(* IEC 61131-3 sources: ml2plc/benchmarks/st (part 22) *)

(* ---- ResNet3.st ---- *)
FUNCTION_BLOCK ResNet3_FB

    (* Model Inputs/Outputs *)
VAR_INPUT
    input_data : REAL;
END_VAR

VAR_OUTPUT
    output_data : ARRAY[0..2] OF REAL;
END_VAR

VAR CONSTANT
    weights_0 : ARRAY[0..63] OF REAL := [-0.190466672, -0.289495766, 0.36445868, 0.11001166, -0.202885658, -0.247976601, -0.217859656, 0.152941793, -0.210685372, 0.322490484, -0.300406843, -0.0737419277, 0.271309823, 0.34986949, -0.269151628, 0.101570874, -0.0975821763, -0.0239237547, -0.28141278, -0.260361493, 0.220720425, 0.342909008, -0.106619239, 0.192217126, -0.139923915, -0.00473925471, 0.256588012, 0.106521919, -0.015166074, -0.237258494, -0.295479923, 0.237283707, -0.111313865, -0.119793385, -0.189164549, 0.109231912, 0.147311017, -0.0809866935, -0.174528345, -0.015255332, 0.110069647, 0.205406636, 0.233189464, 0.175904229, 0.192441761, -0.257080823, 0.113344185, -0.222640619, 0.0253927261, -0.0698330998, 0.304976135, 0.13343668, -0.229343772, 0.317507595, -0.0133918505, 0.251467377, -0.131539866, -0.128968731, 0.204563618, -0.234828115, 0.109687969, 0.0967651531, -0.128085941, 0.0570141077];
    bias_0 : ARRAY[0..63] OF REAL := [0, 0, -0.0451503769, -0.000170675936, 0, 0, 0, -0.0306519736, 0, -0.043658372, 0, 0, -0.0452437028, -0.0463685207, 0, -0.0237470753, 0, 0, 0, 0, -0.0306253415, -0.0182554778, 0, -0.0286273304, 0, 0, -0.0439416394, 0.0359471515, 0, 0, 0, -0.0393987, 0, 0, 0, -0.025377661, 0.0258860644, 0, 0, 0, -0.0256011337, -0.040137399, -0.0210138671, -0.0197667424, -0.0420954861, 0, -0.0343104228, 0, -0.0101194074, 0, -0.0385119878, -0.0309600942, 0, -0.0221530851, 0.0427107885, -0.0482655875, 0, 0, -0.0332414694, 0, -0.0204843841, -0.0293239169, 0, -0.0204854961];

    weights_1 : ARRAY[0..4095] OF REAL := [-0.0287969261, 0.201637134, -0.193626225, -0.0838745981, -0.179824859, -0.158866256, -0.0519343764, 0.0553617924, -0.0298234671, 0.199577436, -0.0565214604, -0.135609776, 0.19474043, -0.0305772722, 0.047594741, 0.174586251, -0.131670237, -0.0606977493, -0.00999130309, 0.160562769, 0.114603773, 0.198183253, -0.0226515681, -0.174445733, 0.0844327062, -0.0653743893, 0.166338369, 0.178600982, -0.179540232, -0.104543671, -0.04106462, 0.0376635343, -0.0928359851, 0.0239627361, -0.0751802325, -0.131423861, 0.107191309, 0.0680955499, -0.134543836, 0.162752822, -0.119452722, -0.118079856, -0.111446388, 0.103158936, -0.0164598525, -0.143377468, 0.0849187821, -0.0122491121, -0.152280733, -0.120597631, -0.0606369525, -0.0807449222, 0.147399679, 0.0629173666, -0.130655468, -0.21262382, -0.169020504, 0.105712339, 0.11746116, 0.0592246503, -0.0597587526, -0.143656209, 0.0653275698, -0.0477767587, -0.154527515, 0.0485876948, -0.0317480415, -0.000382602215, -0.0967821628, 0.0423714072, -0.0512648225, 0.0312831551, -0.17014426, 0.160105124, 0.109350279, -0.0217197388, -0.0921072736, 0.0853802711, -0.0300633907, 0.135347292, -0.0391751528, -0.199345261, -0.195168182, 0.0560685545, 0.215828583, -0.0923638716, 0.192498907, 0.178375289, -0.183688045, 0.116588429, 0.0289125443, 0.0778251439, 0.0613025278, 0.0142809004, 0.0337732583, 0.0574108511, 0.189165697, 0.196946517, 0.107737496, -0.129702166, -0.107477285, -0.107738689, -0.177952528, -0.0559140593, 0.169283316, -0.0538910031, -0.104346119, -0.127213195, -0.0331750959, 0.127317414, 0.0515208095, 0.0195653588, 0.0769012719, -0.124866173, 0.177239373, 0.0280220658, 0.0963039249, -0.0652452409, 0.105720118, 0.15663074, -0.136386782, -0.123085879, 0.0827278346, 0.21160166, -0.16991207, -0.0768297166, 0.120611772, 0.134732291, -0.139711812, -0.184518486, -0.184835598, 0.00858225208, 0.113042273, -0.102391459, -0.0780269504, -0.165388852, -0.140612379, 0.223779544, 0.162238076, -0.00674940646, 0.0487292968, 0.0836367309, -0.19456315, 0.171644017, -0.0955267325, 0.0997560844, -0.0601457544, -0.198954478, -0.00482972385, -0.079228431, -0.127536789, 0.190665379, -0.0999609306, 0.0110752583, -4.10255961e-05, 0.118868679, 0.138081178, -0.0528386459, -0.114722773, 0.170001924, 0.137378082, -0.196978897, -0.15748626, 0.0825704783, -0.033234071, -0.101335384, 0.0289265234, -0.15857622, -0.0556612536, 0.213226333, 0.00719815027, 0.223965615, -0.0638628826, 0.148281991, 0.0975444093, -0.0259753708, 0.0262751374, 0.0979252607, -0.0863377675, 0.0899253041, 0.239503771, 0.289376885, -0.204818711, 0.105383582, 0.293127954, 0.203753337, -0.119700439, -0.16846402, 0.191751063, 0.0327624083, -0.0386312976, -0.264414817, 0.153028056, 0.154591411, 0.124344207, -0.107223384, -0.137165904, 0.0300747007, 0.183606654, 0.198948666, 0.0499654785, 0.144469813, -0.210293442, -0.0324280113, 0.0683567002, -0.04100243, -0.0126516968, 0.164788797, 0.237893194, -0.0847178176, 0.0626023933, 0.155760348, 0.185824335, 0.00780587131, 0.199899733, 0.035005752, -0.0749012083, 0.067025587, 0.141089186, -0.0444214866, -0.0607198402, 0.0990498737, -0.0620695017, 0.0086689936, -0.114031576, -0.111011893, -0.204213917, -0.198096737, 0.138905957, 0.159203395, 0.12167336, 0.0172255039, 0.15101482, 0.131718054, -0.0235928968, 0.200807258, 0.209497362, 0.170748204, -0.231670231, 0.143206522, 0.225486189, 0.104716703, -0.177130625, -0.133289889, -0.0483859442, 0.107198499, -0.0196592454, -0.0476846471, -0.0815907568, -0.135093376, 0.12207596, 0.00658966927, -0.0573140644, 0.0118645504, 0.226763472, 0.178059682, -0.0891532153, 0.0825275332, 0.163484469, -0.0550447851, -0.0375959724, -0.00878846645, 0.0168165267, 0.150091812, 0.084491238, 0.174592748, 0.0785937458, 0.163301513, -0.0316622555, 0.0597050637, 0.157956466, -0.0453870595, 0.101291135, -0.0735865831, 0.0523432046, 0.00310024619, -0.111143999, -0.176621795, 0.0883997232, -0.00594709814, -0.0267459899, 0.164880231, 0.0904007405, -0.00336711109, 0.025017634, -0.136061743, -0.0808758289, 0.139091626, 0.0775778443, -0.155642897, 0.0725118369, -0.0960384831, 0.135437921, -0.188861921, 0.0681308657, 0.121807054, -0.0181216151, 0.126562431, 0.0201322883, 0.0685440749, 0.0470108241, 0.206563786, 0.167886898, -0.182285488, -0.166398615, 0.200898841, 0.191317186, 0.190035328, -0.175405696, 0.124712333, 0.052170679, 0.184364364, -0.0736751109, 0.0639937371, -0.168305129, 0.00677789748, -0.148140043, 0.10284771, -0.13430731, 0.139501527, 0.0359104425, 0.0577303618, -0.188823983, -0.174651235, 0.0696652383, -0.183670074, -0.00257234275, -0.193130046, -0.203748837, -0.153786868, 0.202487156, -0.0460375547, 0.109957233, 0.00299288332, -0.162598059, 0.210710511, -0.194323435, -0.210184813, 0.0554226786, -0.142163336, -0.152110279, -0.0163246542, -0.166943565, 0.175032482, -0.215747178, 0.171988502, 0.132436678, 0.172353908, 0.121031687, 0.186095968, -0.0588158816, -0.0108129233, -0.0942323804, -0.09778703, -0.109081298, -0.106757924, 0.172346756, 0.025905624, 0.0740813166, 0.189657524, 0.148814008, 0.197771326, 0.201267496, -0.068178758, 0.1481594, 0.184583381, -0.014007479, 0.0497234613, -0.0900920182, -0.151112944, -0.154349625, 0.155235782, -0.183371142, -0.164333746, 0.110023871, 0.0927015692, 0.194937959, 0.208203807, -0.00641842186, -0.135277599, -0.0120722651, 0.0209348053, -0.163213924, 0.183399543, 0.00101952255, -0.094531931, -0.0417330861, 0.125320569, 0.140007362, -0.0551816374, -0.0750101358, -0.184187144, 0.0996663719, 0.1298704, -0.00832244754, -0.00248210132, 0.0548401624, -0.0217346549, -0.040534541, 0.0774618536, 0.0789829642, -0.213013336, 0.00969907641, 0.131764188, -0.134339929, -0.16999869, -0.150505453, -0.203993306, 0.133900389, 0.210885063, 0.0592023879, 0.119564161, 0.129766181, -0.116630182, 0.0890186876, 0.0916796774, -0.125102013, 0.144167438, 0.190863922, 0.0828631073, 0.110106811, -0.0818011016, 0.0638723224, 0.0225199312, -0.0798923373, -0.106765099, -0.103232488, -0.0746515393, 0.214082971, -0.139221311, 0.0676382631, 0.20862554, 0.185882255, -0.0279404521, 0.0581518859, -0.0932726786, -0.0684341788, -0.148790196, -0.167229846, 0.160150275, -0.125400275, -0.0166903287, -0.0369179547, 0.0845469385, -0.191490114, -0.161978155, -0.023997426, 0.040678516, 0.14639619, 0.0431083404, 0.0106931906, 0.139329195, -0.149284765, -0.0467167646, -0.0767225027, -0.0320999771, -0.23229675, -0.0372863598, 0.128295347, -0.160325885, -0.148059294, -0.00792731252, 0.0252128541, -0.0963003412, -0.0197790675, -0.0523058102, -0.0141548719, -0.168405354, 0.093509756, -0.0733992159, -0.174149796, 0.0823272243, 0.0543129146, 0.00202205591, 0.112447657, -0.189444944, 0.0949934795, 0.133855537, 0.138600275, -0.170810059, -0.0500965714, -0.186440244, 0.0285257101, -0.000778779387, -0.128126383, -0.0261946935, -0.201500729, 0.11489366, 0.0997269675, -0.138657212, -0.256732196, 0.0291550159, -0.302546233, -0.178278208, -0.234763011, -0.0388856418, 0.0533248745, -0.146624878, -0.0823597312, -0.230229869, 0.0182416849, -0.118736058, 0.0481926613, 0.133541629, -0.114781246, 0.10070549, 0.109701976, 0.0569074266, 0.26510939, 0.00950349867, 0.0546200871, 0.151336238, 0.0048430115, 0.0378029197, 0.144169971, 0.0863773972, 0.200766638, 0.212797061, 0.138086304, -0.182377681, 0.213811055, 0.161403164, 0.124502376, 0.0246564448, -0.196184307, -0.196561068, 0.0875730366, 0.0948206931, -0.149286091, 0.0323978215, 0.0455216914, 0.151648596, -0.127112329, -0.111039624, 0.0246137083, 0.016291365, -0.00267861784, 0.0558695644, 0.201473311, -0.178703129, -0.103530645, 0.173463836, 0.157130465, 0.182277635, 0.0760518163, 0.215445682, -0.106563114, -0.196684077, -0.094135493, 0.10404627, 0.0962792784, -0.0124557465, -0.15429759, -0.0716400295, 0.11189805, 0.0764795393, 0.0549422354, -0.0472201556, -0.00484439731, 0.0528673977, 0.190446272, 0.0174336433, -0.0469030589, -0.0549324602, 0.102302983, -4.00096178e-05, 0.147421315, 0.193782583, -0.0265746713, 0.0705426186, 0.0295248479, -0.134114474, 0.0562623292, 0.172508165, 0.175126389, -0.161904559, -0.0162163712, 0.208393365, -0.100752503, 0.0273437109, -0.153811902, -0.193232462, -0.16940017, 0.188474581, -0.0369768888, 0.0354307853, -0.0991368741, -0.196591377, -0.233054638, -0.118758805, -0.0622535497, 0.0394661725, 0.267733514, 0.107220888, -0.252435923, 0.112368457, 0.166412622, 0.192772374, -0.218732044, 0.126407787, 0.0919501036, 0.00824039057, -0.0796734989, 0.182596043, 0.131103203, -0.109326825, 0.125145733, 0.122357175, 0.0696524829, -0.0965674892, 0.0579061955, -0.200026214, -0.185237691, -0.189040273, -0.224097118, 0.103700139, 0.109744169, 0.283211142, -0.108721465, 0.126635522, -0.0494364649, -0.224469841, 0.151249424, -0.162036136, 0.030354334, -0.00598688424, -0.143472508, -0.047887668, 0.0439753979, 0.0527719408, -0.152598977, 0.110804304, 0.257972151, -0.138091505, -0.110594928, 0.100734361, -0.0214415565, 0.0449742526, 0.22822006, -0.240381643, -0.128085867, -0.0693219751, -0.0846015364, -0.17030485, 0.130928531, 0.00229240954, -0.194736332, -0.0391959101, 0.0145413131, -0.144774944, -0.181710035, 0.032208994, -0.206829414, -0.0198655725, 0.0611966401, 0.00840911269, 0.158986792, 0.126695439, -0.157956257, -0.20029664, -0.104722835, -0.144183606, 0.00487022102, 0.0939430147, -0.0584943891, 0.0557004064, 0.00045491755, 0.114710584, 0.0546646267, 0.20419623, 0.0921241492, 0.0991390496, 0.176430956, -0.158750683, -0.0890071839, -0.179640472, 0.162403598, -0.0909959227, 0.0409451872, -0.0232819319, 0.165903732, 0.069598332, 0.175637826, -0.179648638, -0.00545862317, 0.00749818981, 0.0323755145, -0.158800021, 0.180631563, -0.053162545, -0.014888972, -0.188607126, -0.0488055795, 0.20547007, -0.0377693027, 0.0997820646, -0.124526724, -0.0918210968, -0.167447731, -0.188922942, 0.0540182441, 0.122466967, -0.0612903982, 0.173171565, 0.187880501, 0.0320709199, -0.0716537684, -0.146939963, 0.00549939275, 0.0170418024, -0.156284317, -0.158158392, -0.0161726922, -0.117838174, 0.0458692163, 0.0690316111, -0.102591947, -0.0113369077, -0.0506339818, 0.186475053, 0.10736011, -0.0328097939, -0.13072902, -0.14560762, 0.0873160809, 0.204848334, 0.079661116, -0.018868804, -0.018476963, 0.148941293, 0.0539769381, -0.00221420825, -0.108419128, -0.0766489506, -0.189365566, 0.0919391662, -0.212484032, -0.172094896, 0.0239589214, -0.211048037, 0.189641103, 0.0730664879, 0.206356838, -0.135675371, -0.000756576657, 0.0285059959, 0.209358588, 0.192232445, 0.11306645, -0.115133278, 0.175952092, 0.0211753547, 0.0506318063, -0.19809112, 0.0197272301, 0.054157868, 0.0254253149, -0.155184671, -0.0454918444, -0.196502686, -0.0158347338, -0.135656744, -0.211595923, -0.020885095, -0.00690788031, 0.0370714217, -0.172456279, -0.185076281, 0.160629585, 0.0181837529, -0.0211855043, 0.120963901, -0.00527728582, -0.0352699608, -0.19402647, 0.132209137, 0.0396415927, -0.118135475, 0.00657442212, -0.208759815, -0.0303688291, -0.00777827017, -0.0915059149, 0.11210835, 0.294361055, -0.142053381, -0.0571834072, -0.0146589978, -0.0864291564, -0.101504333, 0.12920031, 0.182926923, 0.192566365, 0.106406614, 0.214629248, 0.06889496, -0.11516425, -0.259321928, 0.184162751, -0.272702873, -0.117973782, 0.0606180206, 0.0292263925, 0.0766455382, -0.120667271, -0.201999113, -0.0266232025, -0.00732299685, -0.0519965291, 0.156876504, 0.123033859, 0.267217845, -0.0109749781, -0.272964209, -0.129237577, 0.053774897, 0.141416252, -0.199857935, 0.0538020581, -0.230259433, -0.0451727808, 0.258897543, 0.148216307, -0.053409934, 0.31615606, 0.0147380829, -0.202499956, 0.110624768, 0.1696845, -0.0922751948, 0.0798982531, 0.0207011886, -0.142718717, 0.0519616678, -0.127546012, 0.126492023, 0.0723542273, 0.147747502, 0.126169741, 0.0813353807, -0.1203655, -0.153749913, -0.0919978395, -0.139003664, 0.0844179541, 0.054092221, 0.110275611, -0.200139761, 0.110008813, -0.126036033, -0.166970596, -0.233972371, 0.0890860558, -0.20025298, -0.230093077, 0.0173213258, 0.275560528, 0.151483357, 0.276097506, 0.00718977815, -0.0111169517, 0.168895632, 0.10235633, -0.240326077, -0.0821303874, -0.00890312064, -0.171553358, -0.00546233356, 0.101003714, 0.0433369204, -0.187788144, -0.103547342, 0.00432489906, -0.109544538, 0.012347714, 0.0869178474, -0.257481515, -0.0600075051, -0.264836371, -0.171154037, 0.0307734851, -0.129194021, -0.199388355, 0.0987441167, -0.0623329841, 0.249395654, -0.034193743, 0.0902072638, 0.203402102, -0.0227374583, 0.0134097785, -0.0912396759, 0.0864051133, 0.0865284353, 0.228083283, 0.126239121, -0.109470509, -0.188946784, 0.00514312088, 0.181860104, 0.0482862443, 0.0316015482, 0.208089277, 0.175173715, 0.157937661, -0.175959155, -0.15175122, 0.0449968129, -0.0724449754, 0.131373897, 0.081098035, 0.0556937009, -0.127380341, 0.131804869, -0.182943538, -0.163977832, -0.00456343591, 0.0986122638, -0.0509269685, 0.144946262, 0.152006164, -0.195760101, -0.158920705, -0.0407915562, 0.0382466763, 0.120302364, 0.163731501, 0.0790192336, 0.0871210247, -0.0502094626, -0.193163037, 0.0618805438, -0.0852957666, 0.124724433, 0.0312432498, 0.114015713, 0.150832668, 0.00696192682, -0.020202592, 0.0919532925, 0.0599388927, -0.155759037, -0.0923569575, -0.0696199685, -0.127464831, -0.187969327, -0.187459841, 0.143950805, -0.0970960557, 0.154307649, -0.05652605, 0.156533435, -0.183348998, 0.139695272, 0.124307856, -0.0476845652, 0.0955802649, -0.0311176628, 0.163419768, 0.113613471, 0.182277307, -0.202524781, 0.0122317718, 0.186174095, -0.113051899, 0.208240613, -0.158425584, 0.0850085169, -0.0775510222, -0.0645689219, -0.0517540723, -0.17061533, 0.0819323882, 0.121917769, -0.119305968, -0.0747042894, 0.0523318127, -0.152910829, 0.100246899, 0.0908019319, 0.066256009, -0.0805988908, 0.0907654166, 0.0451934189, -0.0514816083, 0.192991301, 0.180941716, -0.197929591, -0.0896847397, -0.218640536, 0.058635354, -0.112284772, -0.0678162426, -0.0591657534, 0.190862313, -0.0746522695, -0.0959051773, -0.0859087706, 0.0146463895, 0.127395496, 0.0643470958, 0.222248226, -0.222716317, -0.0038960767, 0.0420699306, -0.189540833, 0.151158154, 0.174533531, 0.0537843928, 0.0724432617, -0.0636890829, -0.0554191582, 0.0796529651, 0.220607117, -0.152003556, 0.0678689852, 0.189509705, 0.196022376, 0.112115934, -0.103596382, 0.0718052611, -0.139615148, 0.17220287, -0.108806856, -0.0700540841, -0.126261801, -0.0981526002, -0.0755177587, 0.112252161, 0.196778193, -0.00826221704, -0.185675785, -0.057513833, -0.101335384, 0.0925282687, -0.0817712694, -0.131041422, -0.0185560435, -0.125542641, 0.191311106, 0.183952644, 0.13196452, -0.153428495, -0.117309444, -0.0829459131, -0.110064179, 0.198635712, -0.171391279, 0.111330763, -0.148759633, 0.0993963033, 0.0926398188, 0.208881006, 0.106514856, 0.205308661, 0.0648586303, 0.000817343593, -0.0404887646, 0.129113868, -0.0304635465, 0.057734862, -0.0244514644, 0.102735177, 0.120236859, -0.138929337, 0.0624369532, -0.155432343, -0.15313834, 0.0859217495, -0.00519438088, 0.126614913, -0.21491994, 0.0207336992, 0.175207987, 0.109249786, -0.054661721, 0.0479473621, 0.00943541527, -0.142473519, 0.116482362, 0.0937203616, -0.0977497622, 0.183454707, 0.126636133, 0.132889017, -0.179818153, -0.00318422914, -0.114538781, 0.190620884, -0.0922307968, 0.171573177, -0.113899581, 0.0264129937, -0.117907241, 0.0159941912, 0.056949541, -0.165546909, -0.079548344, 0.155183807, 0.167912915, -0.12471018, -0.0227756053, 0.195206597, 0.155959591, -0.113060772, 0.0471404046, -0.0937578529, -0.0744760931, 0.0718369633, -0.194636658, 0.0701943189, 0.00457412004, -0.0688510537, -0.159001023, 0.119077131, 0.0420625359, -0.101866595, -0.0260792822, -0.213209078, -0.0761060715, 0.0378767401, -0.0494340956, 0.0950354189, -0.119263433, -0.187393367, -0.19390738, -0.115837008, -0.11679624, 0.0311641246, -0.0763715953, 0.00562612712, 0.104230031, -0.0938740447, -0.158894032, -0.186505824, 0.123571053, 0.0021596998, -0.124141335, 0.0726272911, 0.0728365034, 0.048231259, 0.167245731, 0.173797145, -0.133879036, 0.123410001, 0.0136341602, 0.211613938, 0.0339705497, -0.0568555892, -0.0638442487, -0.165108442, 0.113140717, -0.114156596, 0.0502677411, 0.105490163, 0.154489145, 0.0633081943, 0.0605547279, -0.168472469, -0.174018279, -0.178102687, -0.0923157632, 0.0868086368, 0.142751232, 0.0472065359, -0.0355895907, -0.070602119, 0.0226132125, 0.111900166, 0.072677359, 0.126415685, -0.147081137, -0.145128071, 0.119609222, -0.149196088, -0.0602950752, 0.198493585, 0.137908891, 0.0641960949, 0.200968578, -0.0566390008, -0.1688862, 0.172993645, -0.144077167, -0.197343826, -0.0247414112, 0.199622199, -0.1655339, -0.0133733898, 0.134934023, 0.0719420165, 0.000706866384, 0.149509206, -0.156804532, -0.0837745517, -0.037465632, -0.157091066, 0.107307032, -0.00644093752, 0.0704480559, -0.183203697, -0.196138009, -0.117853299, -0.12040215, -0.11014574, -0.116727851, 0.026737988, -0.0404386818, 0.0639270395, 0.104571596, 0.0609508008, -0.0830935389, -0.20587337, 0.0998597592, 0.0920080096, -0.113937676, -0.0127168447, 0.130367443, -0.162072524, 0.206473872, -0.0470631719, 0.202682182, -0.0224076658, -0.0183282048, -0.0392407626, 0.13104786, 0.0124193132, -0.155867845, 0.187796101, 0.12736474, 0.183426574, 0.0451046377, 0.0507078916, 0.122980073, -0.21496205, 0.0355659574, -0.0358312726, -0.136690676, -0.167069823, 0.0553592891, 0.212405875, 0.186634675, 0.140052691, 0.0532232374, -0.132964134, 0.199990019, 0.129920498, -0.0277204067, 0.162883624, 0.197279349, -0.0547595471, -0.169750974, -0.0363512784, -0.0266377479, 0.122363672, 0.0337654799, -0.199149102, 0.207519457, 0.142926887, 0.215468749, -0.0605023801, -0.0568595082, 0.0636674613, 0.106427982, -0.139160648, -0.11427062, 0.189653918, 0.135131165, -0.0713291317, 0.103454813, 0.115515873, 0.0241415501, -0.141884476, 0.0647414476, 0.1221935, 0.187437966, -0.0765461177, 0.130906656, 0.209548905, 0.198075101, -0.0151947271, 0.106877655, 0.122374028, 0.0876808092, -0.0646020845, 0.179015324, 0.137440547, -0.111645944, -0.0637109131, 0.264909327, -0.00986942649, 0.19460775, -0.215875, -0.216673881, -0.195247158, 0.0369132459, 0.22958532, -0.0758189484, 0.161118656, -0.0532057211, -0.111272402, 0.0191001799, 0.154950529, 0.184459001, -0.0586241372, 0.211076126, 0.0385005176, 0.0375854224, 0.185866401, -0.0925790668, 0.0594946295, -0.199379593, 0.160706773, -0.0215413142, 0.0920865387, -0.0727619678, -0.0503336526, 0.144037127, 0.0390647538, -0.176736578, 0.218084648, 0.282077163, 0.0684015825, -0.0997406542, 0.0936136246, -0.0177756548, -0.116294734, -0.21881853, 0.0861533135, -0.144913971, -0.116913833, -0.228465006, 0.243279889, 0.289645553, -0.157389015, 0.0694431514, -0.0845005885, -0.169205248, 0.0732500702, -0.140289873, 0.217532694, -0.153820172, 0.165036872, -0.0370052084, -0.0649239048, 0.00705603603, 0.00300642545, -0.147408083, -0.0400309153, -0.0219824761, 0.021092033, -0.0739108026, 0.0152327912, 0.16345866, -0.169258162, -0.171906739, -0.0344251506, 0.0626144186, 0.0827743858, 0.0153012248, 0.214705959, 0.149533838, -0.0852295235, 0.108769022, -0.125927284, 0.0506657287, -0.0685000271, 0.132542357, 0.189130142, -0.107204311, 0.208437741, -0.0613691844, -0.15225552, 0.0756992996, -0.0966535062, -0.198031753, 0.0743363649, 0.0633449629, -0.129061252, 0.122365281, -0.130634353, 0.0883900598, 0.0156343877, -0.135135397, 0.198845685, 0.2392952, -0.145629406, 0.188295275, -0.13789998, 0.132967234, 0.132922307, -0.17668727, 0.245915323, -0.141065955, 0.192191795, -0.157576233, -0.085805878, -0.0276803467, -0.095566079, 0.219359696, 0.202878788, -0.0802682042, -0.176504254, 0.023325054, 0.0037062054, -0.138832927, 0.053536851, 0.127934501, -0.168392971, 0.0300281346, 0.0400527865, -0.206524342, -0.081766516, 0.104110494, 0.00106944144, -0.120554268, -0.0580964088, 0.109146222, -0.000105708838, 0.182546988, -0.148469537, -0.148119092, 0.149815395, 0.205082461, -0.0108131766, 0.179644182, -0.192448467, -0.0218183249, 0.112928316, 0.173357442, 0.0719634742, 0.20145084, 0.0719409138, -0.164568782, -0.130916566, -0.202400431, 0.0947056264, -0.192789838, 0.0868111402, -0.00978286564, 0.196489051, -0.0734990388, -0.146960199, -0.000552743673, 0.0167299211, -0.199335337, -0.158682853, 0.0911645144, 0.180834278, -0.122386955, 0.00548417866, -0.187905684, -0.107697234, -0.084947437, 0.0716611892, 0.132587507, 0.13105391, 0.0321043134, 0.0708666295, 0.136131003, 0.0918786675, 0.0526147634, 0.14389886, -0.0311155468, -0.188370556, -0.212843508, 0.0522523373, 0.167048857, -0.206337899, 0.072918728, 0.120494351, -0.190175474, -0.154683962, -0.000773754495, -0.186758995, 0.25392881, 0.165069968, -0.174278378, -0.0480074361, 0.0444551259, -0.0307127461, 0.197782025, 0.127323076, -0.19140029, -0.17637898, -0.0651647598, -0.0631855875, -0.170364678, 0.128072217, 0.142127141, 0.0896252617, -0.168872684, 0.0608825311, -0.199593708, 0.0163794793, -0.111544512, -0.0925613791, 0.0456584245, 0.273554981, 0.0908730105, -0.121767685, 0.133312061, -0.0430089869, 0.048706051, -0.106118105, 0.156891361, 0.199550763, 0.0661296993, 0.190545216, 0.0400548801, 0.0303085539, -0.0425427854, 0.0662297159, 0.266184568, 0.028025724, -0.122740746, 0.0264457632, 0.00358478306, 0.129521757, 0.162871301, 0.26886633, -0.0782814473, -0.0386863798, -0.0817479417, 0.0508834422, 0.212506562, -0.104619637, 0.0130023751, 0.0292652808, -0.08503066, 0.158758327, 0.0168799069, -0.0856374726, -0.150301456, -0.0860033929, -0.118447781, -0.179989219, -0.0929494426, -0.0466621518, -0.0659421533, 0.121023342, 0.105154112, -0.0455614179, -0.203972697, 0.173838392, -0.0386415124, -0.0278328806, 0.178764507, 0.104911312, 0.108715996, -0.0253986865, -0.168122798, -0.114805967, -0.0621888191, -0.0132009238, 0.0253832936, -0.0265160799, 0.0423865467, -0.100953348, 0.172172591, 0.201425806, 0.141991392, 0.0940631181, 0.194293097, 0.0401813537, 0.12128751, 0.196684197, -0.0543928444, 0.0463825911, 0.0403407067, -0.21529898, 0.00518736243, -0.0455965251, 0.0162204355, -0.183138445, -0.193831608, 0.187192395, 0.00752931833, 0.157815233, 0.141796991, -0.0405156463, 0.198203638, 0.00560341775, -0.0508095473, -0.0763344318, -0.0735320747, -0.0695720166, 0.148685709, 0.0700013191, 0.182473376, -0.1108841, -0.0968367755, 0.0362190455, 0.036774829, 0.0170685947, -0.0752303004, -0.0852943808, -0.206426427, -0.149846435, -0.155158252, 0.119575307, 0.0180834234, 0.146422639, -0.101406202, 0.0536810011, 0.0994656831, -0.0630992353, 0.0158559978, -0.0455258042, -0.21185334, -0.118426792, 0.159210399, -0.116417825, 0.0386347026, 0.159501418, 0.033601746, -0.0757299215, 0.00185963511, 0.085397765, 0.083639726, 0.178043649, 0.190545216, -0.0945898443, 0.0499521047, 0.0201606303, 0.106833711, -0.0188183188, 0.177461788, -0.100810207, -0.0469589531, -0.0987466872, 0.177121416, 0.1593398, 0.0223871171, -0.208162114, 0.062356934, -0.125736207, 0.096315518, 0.0971169025, 0.0245347768, -0.020675838, -0.111754142, 0.212888882, -0.170801476, 0.0786470622, -0.0122303218, 0.162038699, -0.199096397, 0.170362726, 0.0747093409, 0.111208364, -0.0473197848, -0.0435504466, -0.0453317761, -0.110917084, -0.0126232058, -0.177978754, -0.0992414504, 0.130278543, 0.018110469, -0.0700823665, -0.114136361, 0.0361899287, -0.18268013, 0.0165710393, 0.0793500915, -0.00841967668, 0.125138253, 0.0887469351, -0.107942894, -0.239920467, 0.201740548, 0.149393812, 0.203771755, 0.0577221662, -0.00337263942, -0.146427289, -0.257600576, 0.119674787, 0.194880754, 0.245413616, 0.0804518312, -0.166380689, -0.000451727072, 0.0460289009, 0.132229939, -0.1964733, 0.187092066, -0.0433319323, -0.0352629423, 0.137847543, 0.182559997, 0.0790997595, 0.114835717, -0.0771531537, -0.0737332329, 0.0758020729, -0.0452585854, 0.145568117, -0.1918246, -0.0583546832, -0.0145606585, 0.129812345, -0.0127620762, -0.0558166765, 0.16816707, -0.0112826349, -0.0819175765, -0.239855021, 0.103059068, -0.215481281, 0.116379917, 0.0303741544, -0.0232816786, -0.142835721, -0.178205758, 0.208591044, 0.288504571, 0.160375908, -0.10488455, -0.0112059414, 0.149956122, 0.0636754483, -0.195255071, 0.108991124, 0.206127957, 0.259172261, -0.150578156, -0.0045624678, -0.199588045, -0.115991615, 0.0703731775, -0.22166048, 0.115133122, 0.07192339, -0.00083938241, 0.0757085681, 0.160763949, -0.0662796795, -0.172549099, 0.0753220916, 0.121819116, -0.186484084, -0.165406242, -0.0917130634, -0.127552748, 0.209713519, 0.00541543402, 0.108752683, -0.048205357, 0.210129693, 0.0972502008, 0.211364299, 0.0602482185, 0.123633213, -0.154390544, -0.117387019, 0.105454966, -0.0183485299, 0.154096812, -0.168688595, 0.0630255491, -0.190940425, 0.13162984, 0.201842621, -0.189648613, -0.0979222134, 0.0130105121, 0.00230050553, -0.157333851, 0.13677448, 0.0410381854, 0.0108493455, -0.126054719, 0.0934812054, -0.0121305455, 0.150938109, -0.197522938, -0.216986924, 0.12068636, 0.100021429, -0.0908799618, 0.168728262, 0.0442929193, 0.139804959, 0.00512484135, -0.041490376, 0.163413405, 0.122350357, 0.0158086959, -0.161861941, -0.0287991706, -0.0309194028, 0.180298939, -0.0883494616, 0.163443282, 0.213652179, -0.0104613453, -0.0396695137, 0.153360203, -0.148807853, 0.00914561749, -0.165651739, -0.1075399, 0.120668754, 0.15019466, -0.168916598, -0.159659475, 0.134091392, 0.13391538, 0.0127349049, -0.148728609, 9.60677862e-05, 0.0587041825, -0.114760749, 0.076023981, -0.198310554, -0.122234218, -0.00825509429, -0.196786553, -0.111470282, 0.0473584384, 0.0859691352, -0.0197229534, -0.139441609, -0.195919603, 0.214953706, -0.211334214, 0.0864942521, 0.149090514, -0.0995983481, 0.14995639, -0.211273924, -0.128281027, 0.134673044, 0.206308767, 0.173526242, 0.00177001953, 0.178798303, -0.186740786, -0.125183105, 0.190860763, -0.15597181, 0.104340389, 0.0919784755, -0.109020695, 0.123255745, 0.160754845, -0.0181522816, 0.00826106966, -0.108122781, -0.118333563, 0.0240668505, 0.0728541166, -0.0888753533, 0.0701249689, -0.0911424607, -0.035492748, -0.0625108778, -0.201834172, -0.00986467302, -0.171905458, -0.198220938, -0.125818759, -0.0823892057, 0.124080285, 0.133759275, -0.0294942409, -0.023840189, -0.166492149, 0.0786484629, -0.0805669874, -0.202838793, -0.0324053615, 0.161780253, 0.125890866, 0.162339553, -0.184726253, 0.0838932842, -0.0687282532, 0.192603484, -0.0388252288, -0.127744973, -0.213563338, -0.101094738, -0.00717841089, -0.0166087151, -0.203627214, 0.183910921, 0.00717809796, 0.12827535, 0.0516086072, -0.162369341, 0.120600984, 0.186384007, 0.0617960542, 0.115706041, 0.115686163, -0.0111425072, 0.120042011, -0.0624903291, 0.010419935, -0.0645890683, 0.128529057, -0.0571770221, -0.175542116, -0.0534045845, 0.154075637, 0.0780510157, 0.0838643163, -0.127966419, -0.0523578525, -0.163016126, 0.00269818306, -0.0729043931, 0.213392332, -0.0667243898, -0.00207157433, -0.0347132534, 0.0671278983, 0.0825990885, -0.176288694, 0.115147576, 0.144309029, -0.0388330817, 0.0370965153, -0.145275503, 0.115442678, 0.137224212, -0.0672999918, -0.0209041983, -0.0843738467, -0.076107353, -0.13899076, 0.0134440958, -0.106940709, -0.0790602267, -0.100989997, -0.0825085938, -0.0422780812, 0.216143265, 0.0434457213, 0.171689466, 0.0899863094, -0.00309301913, -0.0964013189, 0.0696323663, 0.11887081, -0.0692265779, -0.194193363, 0.121454194, -0.191472918, -0.110765375, 0.0960554034, -0.101598121, 0.114441469, 0.0659235865, 0.130200818, 0.121813938, -0.0578708351, -0.086437434, -0.108647905, -0.0607499927, 0.0430828184, -0.193046167, 0.0327921957, 0.0684836358, -0.186204255, -0.183985829, 0.110593989, 0.0532316118, -0.177710846, -0.163656503, -0.173432246, -0.0314968079, -0.151612878, 0.143427029, -0.165966004, -0.0755198747, -0.208826602, -0.17920956, -0.0773960352, 0.0872260183, -0.0976994857, 0.114518069, 0.110299453, -0.0676979423, 0.206201911, 0.056230519, 0.158488706, 0.0116583984, 0.152704671, 0.0783563405, 0.197553605, -0.184350356, 0.189391062, 0.0166197326, -0.0901755169, -0.191783831, -0.118035868, -0.0449252799, -0.0107128965, -0.0816708133, -0.0544931963, -0.204584405, -0.0387687087, -0.0949772447, 0.0460221358, -0.000431137101, -0.173131198, 0.0689009875, -0.0812623948, -0.190199226, -0.160632268, -0.150214508, -0.0479303226, -0.133730575, 0.12269488, 0.132861421, 0.116756126, -0.0625272542, 0.0453324765, -0.212504029, -0.180632263, 0.229810223, 0.0990021825, -0.195593789, 0.235955507, -0.249435619, -0.192426175, -0.0116430558, -0.22546199, -0.0619180687, -0.0813810825, 0.178630605, 0.0092575727, 0.176159397, 0.298030823, 0.185510695, -0.137530193, -0.0452765115, -0.207549289, 0.146510646, -0.171670303, 0.265041798, -0.0187018663, 0.135485336, -0.129769668, -0.193181783, -0.213981807, 0.192192391, 0.147625938, 0.156314656, 0.05699341, -0.142236948, -0.119077913, 0.179841056, -0.0629975945, -0.104762428, -0.125211447, -0.14266631, -0.0601936877, -0.0364018083, -0.0799863786, 0.0712708384, -0.181263745, 0.128054276, 0.0881264061, 0.0278715938, -0.0938142166, 0.108250186, -0.0280871093, -0.173671246, 0.154439613, -0.199859276, -0.207510322, 0.113391146, 0.0949654132, -0.157867059, 0.0300325751, 0.0347745866, -0.0836828798, -0.109618604, -0.0289660841, -0.202263281, 0.21372427, -0.105892681, 0.191544786, -0.170336902, -0.150212094, 0.197368309, -0.186274111, -0.170028225, -0.00803947449, 0.194047078, -0.0991749167, -0.119580686, 0.0488605946, 0.0256551802, -0.125362441, -0.0738906264, 0.206044659, 0.00442288816, -0.175227448, -0.152266279, -0.199678972, 0.0752449185, 0.0161459446, 0.208508387, -0.198326081, 0.0312630236, 0.174753115, 0.153398082, 0.140059993, 0.0729063898, 0.174086884, -0.0703520328, -0.195192233, -0.157076001, -0.036226362, -0.205104709, -0.174567297, 0.0171607882, -0.116198495, -0.0708719939, 0.044384256, -0.159294024, -0.13956818, -0.147202596, -0.172137842, 0.0154579133, -0.0588126779, 0.155877337, -0.0972540677, -0.0985946134, 0.108118966, -0.0442180336, -0.0142957121, -0.113704823, 0.0837571472, 0.0825636238, 0.100469217, -0.193166032, -0.189904317, 0.110404596, 0.111059561, -0.0263882726, 0.0777775496, -0.194304436, -0.132153511, 0.118601069, 0.0515244752, -0.0868103802, -0.092175208, 0.182618186, 0.0733394772, -0.110395521, -0.153526604, -0.0347853154, 0.129671916, -0.140404195, 0.10624896, -0.198270962, -0.146404207, -0.206243992, 0.176455781, -0.125557557, -0.192070216, -0.0227239877, 0.213343993, 0.128212437, -0.0822850317, -0.155388311, -0.0103898495, -0.119988322, -0.00629195571, 0.0263843983, -0.0645047724, -0.131128609, -0.0325913876, 0.135626957, -0.072056964, 0.0038716346, 0.195447132, -0.211576611, 0.000806346536, 0.142347768, 0.193100467, -0.204855338, 0.00235620141, 0.0648757964, 0.205600873, 0.13106589, -0.0140479952, -0.196146876, -0.132513404, 0.145923689, -0.13448292, -0.00566205382, 0.185168788, -0.09505447, 0.0785790831, 0.0351739079, 0.205144569, 0.137520716, 0.16661109, 0.196318254, -0.213474959, -0.0414532572, 0.103707328, 0.0494590253, 0.0121845901, -0.14195092, 0.168113038, 0.106775209, 0.00271753967, 0.0252564102, 0.122725263, -0.0311934501, -0.200210854, 0.131448641, 0.205436215, -0.14131099, 0.0286722034, 0.168602541, -0.047244519, 0.0403911918, 0.13908349, 0.0185234249, -0.117879212, 0.0941817015, 0.170137122, 0.0652392656, -0.0828565061, -0.0910385549, 0.177681938, 0.102450922, 0.0477524549, -0.163797021, -0.101946861, -0.214260817, 0.0238904785, 0.225524053, 0.208094507, 0.0252908356, -0.174766853, 0.010269451, -0.0447409302, -0.0171606299, 0.0435046591, -0.211344436, 0.137196705, -0.00548750954, 0.106041424, -0.03372702, -0.0689889714, 0.176017016, 0.0693399906, -0.0631261542, 0.0570853353, 0.110590167, 0.158552811, -0.218137234, 0.227292344, 0.228224993, 0.104598656, 0.191354856, -0.0603202321, 0.0390501469, 0.160037979, -0.0421753563, -0.012174543, -0.0599781871, 0.0374898314, -0.16964066, -0.0145777613, -0.150289029, -0.222676113, -0.130118147, -0.0851336271, 0.0560929105, 0.124441281, -0.0389688611, 0.211753815, -0.3047176, -0.195135519, 0.0575269051, 0.118676692, 0.254068643, -0.0964110196, 0.103781089, -0.0195431523, -0.00197520107, -0.0391661637, -0.0210434217, -0.0949213803, 0.0830372572, -0.200275943, 0.184665754, -0.0754128322, -0.108697027, -0.194729984, -0.0860964432, 0.163379699, 0.195537135, -0.220752254, 0.183663502, 0.0367836021, -0.193053201, -0.213411212, 0.169405296, -0.210496545, 0.089611128, -0.0914427266, -0.146663666, 0.112126216, -0.190471187, -0.151629761, -0.118191868, -0.161780074, 0.0700828135, -0.023731539, 0.0662216842, 0.0570927225, 0.151051804, -0.0581127815, 0.187727496, 0.164582342, 0.108500071, 0.0806025043, 0.132105574, 0.171909839, 0.151336297, 0.0216216911, -0.19720386, -0.0865775421, 0.0918769985, 0.0651388541, 0.101763561, -0.165228412, 0.0967422575, -0.197852328, 0.0326667093, 0.149067357, -0.202845722, -0.0753694028, 0.185080975, 0.112593286, -0.0308894385, 0.146897539, 0.139629066, -0.0057492801, 0.196031645, -0.0433132499, 0.0949817896, -0.22793296, 0.140323445, 0.20535101, 0.00654665194, 0.0543287173, 0.082761243, -0.0949113667, -0.19657506, 0.0682489723, 0.184988469, -0.0549624749, -0.155943945, -0.159202754, -0.000955834985, -0.0745041221, 0.0357825309, -0.0457972139, -0.0863496214, -0.068731755, 0.156966105, 0.102031305, 0.0772381872, 0.0516668707, -0.069934696, -0.171752036, 0.0247167349, 0.197206363, 0.000397771597, 0.0669030994, -0.0112306774, 0.121345595, -0.181874871, -0.102461353, 0.130182162, -0.0321843177, 0.0372402221, -0.0465781689, -0.18494001, -0.0399046838, -0.0770143121, 0.134995177, 0.189494893, 0.148261294, -0.061371848, 0.119698837, -0.20221296, 2.30669975e-05, -0.205027491, 0.0951066166, -0.168831587, -0.0747900307, -0.121398196, 0.178700998, 0.0287471116, -0.0423051268, -0.106853776, 0.205980286, 0.215550825, -0.0599444807, 0.188939258, -0.098034136, 0.0424312502, 0.113852099, 0.00394080579, 0.0708767325, 0.0387572497, 0.193161801, -0.105255395, -0.149511009, -0.183171943, 0.0543221086, 0.000958368182, -0.0319679826, 0.089403823, -0.011545077, -0.0130462199, 0.00551834702, -0.00398561358, -0.0225462615, 0.157178923, -0.204262495, 0.022420153, 0.00691081583, 0.202832952, 0.103284314, 0.0576447994, -0.168464258, -0.160268232, -0.16031602, 0.13101922, -0.102683522, -0.0796382576, 0.0150442421, 0.057686463, -0.00462538004, -0.0570764691, -0.112117276, -0.202424645, 0.177651122, -0.060906291, 0.14917542, -0.0663579404, 0.207064077, -0.0621602237, -0.0727250576, -0.0505298674, 0.166853115, 0.131181166, 0.0528817028, 0.182591543, -0.131295085, -0.214916736, -0.167643577, -0.171931058, -0.0976076052, 0.0673984438, -0.192280039, 0.160496429, -0.096597679, 0.0677601844, -0.0665755719, -0.0466447473, -0.134645581, 0.0446114689, -0.188451454, 0.065866366, 0.0944281369, -0.0774573982, -0.128453493, 0.084732458, -0.0828902125, -0.0460760146, 0.0562799424, 0.0572096854, -0.120285958, -0.0611797273, -0.0863713622, -0.0313139707, -0.158191442, -0.0913565308, -0.0547137558, -0.0715128481, 0.148597136, 0.0647662133, 0.0948180407, 0.1016884, -0.107101806, 0.112274364, 0.130645767, -0.132742882, 0.063240245, -0.0239790529, 0.214894965, 0.039905265, -0.166711584, -0.164006442, 0.00362469256, -0.0177395344, -0.142894775, -0.0920766145, 0.0557132512, -0.105091035, -0.0341222584, -0.126966149, 0.0203460455, 0.194955453, -0.0237233341, -0.049101457, 0.0987512916, -0.188197687, -0.00309565663, -0.0618091077, 0.121471658, 0.114097014, 0.0614005476, -0.0874201059, 0.118369386, 0.0488611311, -0.0974244624, 0.060956791, 0.09975712, -0.0146490484, -0.213436767, -0.116138719, -0.0667345077, -0.209338829, -0.196749538, 0.202766106, -0.122498922, -0.212087691, 0.21396865, 0.0765298456, -0.0631021708, -0.114263915, 0.137899652, -0.0875501335, 0.0651765019, -0.172441825, 0.0399881452, 0.0264455229, -0.148256093, -0.208674431, 0.0328289419, 0.0215819627, 0.0447034687, 0.0569855124, 0.0466875732, -0.154296696, 0.0557099953, 0.099412255, 0.0885903686, -0.138083339, -0.215496168, 0.0766443089, -0.029674679, -0.159911841, -0.193334565, 0.129661992, -0.209483698, 0.0277790427, 0.0214523505, 0.125006989, 0.206167772, -0.247479483, 0.110709831, -0.0240806229, -0.106150419, -0.0156477932, 0.23906444, 0.0239258539, 0.0397250541, 0.159573585, 0.0976805016, 0.028400287, -0.184984565, -0.135613933, -0.235051349, 0.158971772, -0.100035571, 0.098122105, -0.0841649026, 0.181454465, -0.190613255, 0.126531929, -0.0978783965, -0.0936749801, 0.0890369713, -0.0226638466, 0.0344321169, -0.231752813, 0.125484258, 0.0367094986, -0.177370921, 0.217156366, 0.190573201, 0.178353146, 0.0782344341, 0.197666898, -0.0849834532, -0.117577732, 0.130946651, 0.117060021, -0.171168283, -0.0270178616, 0.169972658, 0.210708454, -0.176258653, 0.241882116, -0.0276549459, 0.0397499725, -0.12462277, 0.0972123072, 0.289701581, -0.09509027, -0.195481196, -0.0970052183, -0.0570235103, -0.230527118, 0.168534026, 0.0795216113, -0.0857440829, -0.104283124, 0.0783484355, 0.0913527161, -0.175007626, -0.0441816524, -0.101990119, -0.0751975626, 0.0174092911, 0.0910891965, -0.072370857, 0.0863547698, 0.030440174, 0.0699474886, -0.069681555, 0.244500011, 0.132901147, -6.72638416e-05, -0.011448239, 0.0668040514, 0.0330525972, 0.0399980098, -0.0805684775, -0.0893881321, 0.00371935964, -0.089494504, -0.135875374, -0.00690581929, -0.0437228978, -0.139606163, 0.138900653, -0.189150035, 0.0839610398, 0.064339444, -0.219201058, 0.10751234, -0.138615251, 0.25648123, 0.193666056, -0.195941389, -0.0475867949, 0.170852602, 0.0483538099, -0.23815763, -0.215300962, -0.0604494624, 0.157071248, -0.198099524, 0.1605075, 0.187679827, -0.110149607, 0.260497242, 0.0667465031, 0.0740663335, -0.0811945647, -0.0274696928, 0.256537765, 0.112993523, -0.176565573, -0.211348012, -0.174424976, -0.0731801093, 0.107577667, 0.137092873, -0.183942825, 0.161429822, -0.234576806, 0.153691486, -0.0336565897, -0.0619529299, 0.1576882, -0.00832078699, 0.144546583, -0.0621412583, 0.0572977401, 0.0700711533, 0.107443564, 0.247199208, -0.107651167, 0.257766634, 0.212229684, 0.0449296683, -0.0885326862, -0.01169773, 0.0446972661, 0.132320687, 0.146239325, -0.125418752, -0.0602291077, -0.145199999, -0.0226940326, -0.042851422, -0.200135052, -0.0707998723, -0.0483647697, -0.0434840582, 0.0195474084, -0.0806870908, -0.066419743, -0.0243462902, 0.187009096, 0.266266257, 0.0210534781, -0.190431267, 0.0193590894, 0.0430474356, 0.0968303457, -0.0600356534, 0.212457985, 0.0733742341, 0.0564355701, 0.00829766691, -0.0975096449, -0.0297273509, 0.0435266942, 0.232403845, 0.175813645, -0.0605938882, 0.075977318, -0.102545507, 0.159124359, -0.0323878899, -0.11937844, -0.210411832, -0.0369421095, -0.0605836548, 0.0146844471, -0.162964344, -0.180745065, -0.138387382, 0.191610858, -0.0805439204, -0.0106778275, 0.195784792, 0.140448511, -0.108700931, 0.154517576, -0.139445692, -0.0971742496, -0.156008646, 0.0350373723, -0.00932324678, -0.0389326066, 0.157756582, 0.0591719672, 0.191582471, -0.109771289, -0.205349728, -0.123457506, -0.113767751, -0.199369431, -0.0199184865, -0.0721435249, 0.0268921331, 0.17901054, -0.0615942702, -0.196627244, -0.0978841856, -0.0243181754, -0.252508283, -0.171970218, -0.00553819537, 0.138990164, 0.176095605, 0.0951418132, 0.00899968576, -0.21385926, -0.197060034, 0.193683833, 0.233065248, 0.06070612, 0.0120316064, 0.0260351393, -0.0639142916, 0.173514277, 0.204962239, -0.202115402, 0.188184857, 0.059859708, -0.160158709, 0.194068417, 0.03272672, 0.0373210721, -0.154273242, 0.192293808, -0.200334892, 0.123418614, 0.0633706972, -0.0923486948, 0.114942677, 0.198776662, -0.215897352, 0.0565530509, 0.0895846412, -0.13462013, -0.0126579404, -0.177565232, 0.158671334, 0.233714014, -0.193006068, -0.281954676, 0.156786814, 0.144733921, 0.151347488, 0.173282146, 0.276410073, -0.19197917, 0.292017668, -0.151239187, -0.149175525, 0.0274241325, 0.188164338, -0.293288738, 0.0220334232, -0.273543179, 0.0642050654, 0.08832784, 0.134583443, 0.0807607248, -0.000400550896, 0.0918587297, 0.07559672, 0.314674675, 0.0490694642, 0.101967268, -0.241429016, 0.0202955063, -0.209007189, -0.106268622, -0.0069014011, 0.10103409, 0.0636226386, 0.0471041873, 0.000416273368, 0.26530841, -0.10846144, 0.142565444, 0.216730133, -0.137502536, -0.120941207, 0.180886477, 0.118575349, -0.0189697742, 0.239887834, -0.142993346, 0.146749064, 0.187433407, 0.0744013041, -0.0447228253, 0.205760106, -0.0467358679, 0.0100782812, 0.180402741, 0.0978421122, 0.068239525, 0.164465442, 0.00975632668, 0.195215091, -0.0487101376, 0.0192688555, 0.031739369, 0.199693933, -0.0508198142, 0.123593971, 0.0872715563, 0.148543522, -0.150334686, 0.0227344036, 0.115462556, -0.0487159789, -0.016429022, 0.0369556397, 0.0111047179, -0.0476019233, -0.118862145, -0.0377347171, 0.0323484689, 0.0822030753, 0.0403838307, -0.0443079621, 0.0296327919, 0.104416624, -0.03586936, -0.162577927, 0.140675917, 0.0654677302, -0.155557871, 0.0191291273, 0.213035539, -0.174402893, -0.124022201, 0.169056132, 0.158662096, -0.163972616, -0.0827359259, -0.00124819577, 0.010516569, 0.212345287, 0.0464865416, 0.110000417, -0.154047757, -0.0204191953, -0.08001028, 0.064174667, -0.212888524, 0.0529602021, 0.211512908, -0.190684035, -0.0921802148, -0.151814789, -0.00803656224, -0.00784375705, -0.141917571, -0.00132001087, 0.0526149124, -0.136854231, 0.0130218118, 0.0680401698, 0.0399013944, -0.186063141, 0.0169487298, -0.0813166797, 0.116694055, 0.042951867, 0.0821733102, 0.134713322, 0.184491575, -0.191935867, 0.0131632471, -0.100137152, 0.182891071, 0.000961091835, 0.12456546, 0.145593375, 0.00720275845, -0.105598301, 0.207914561, 0.00380734471, -0.0248022173, -0.160123363, 0.0381194986, 0.129718468, 0.123341523, -0.0176308304, -0.175096646, 0.110144205, 0.0652518645, 0.094259724, -0.0674603283, 0.224985868, -0.048998557, 0.00546664651, 0.0410965495, 0.107289985, 0.00302270707, 0.0922987014, -0.0397922322, 0.0962653086, -0.093549408, 0.048931852, -0.0534424298, 0.0138503471, -0.0754063874, 0.065585278, -0.0900662616, 0.139983714, 0.128798306, -0.0214835256, -0.0355337039, -0.00254588644, -0.0779585242, -0.10749051, 0.0774092972, -0.195456222, 0.203156188, 0.103489295, -0.0295414776, -0.0359847844, -0.132312894, 0.139603063, -0.0406532735, -0.114045464, -0.155046389, -0.111411333, 0.0317999125, -0.166794747, -0.167081028, 0.0591999739, 0.129730806, -0.175916776, -0.0256558955, -0.0691830069, -0.0288138986, 0.0313598067, 0.0193842202, 0.0408626944, -0.172637001, 0.0734120756, -0.202827275, 0.190578565, 0.153090999, -0.0792387873, -0.00259576738, -0.0505202115, -0.212944731, -0.159402311, -0.0976085365, -0.0191448629, 0.130320415, -0.0283066481, -0.0278123319, 0.00982235372, -0.0937846899, -0.162156463, -0.143455982, -0.00604511797, 0.0269212872, -0.194088265, 0.10351716, 0.00833112001, -0.0464727581, 0.129887775, 0.046137765, -0.183257371, 0.0989542454, 0.0501036495, -0.156223819, 0.0834358186, 0.128036156, 0.00859726965, -0.0364925116, -0.197799727, 0.164447352, -0.122780189, 0.000409752131, -0.0851694047, -0.127068669, 0.124540463, -0.0155066447, 0.220182613, 0.0643692538, 0.0083350027, 0.208433077, -0.083687149, 0.139471397, 0.0637006313, -0.166873068, -0.044224903, -0.152341023, -0.0996580869, -0.00282181404, 0.0116580725, 0.0610121377, 0.153579026, -0.151627228, 0.0830854848, -0.0748153627, -0.00402663695, 0.196929038, 0.199087873, 0.162471503, 0.103831865, 0.0201131664, -0.0360102542, 0.155990794, 0.104891919, -0.0791717842, -0.173016161, 0.0897792131, -0.0222959071, 0.011724811, -0.0878165364, -0.0617964715, 0.103893965, 0.117816001, 0.046961911, -0.0394895524, -0.172319263, 0.0261968896, 0.128624946, 0.000213261112, 0.096357584, 0.183724195, 0.0663415045, 0.128639147, 0.257106632, -0.126175031, -0.166864216, 0.0406238586, -0.0439073667, 0.234832495, 0.110920966, 0.147819847, -0.0325478055, -0.145270362, 0.123860314, 0.0187417157, -0.133771777, 0.0191091448, -0.018727826, -0.212830409, 0.0778542906, -0.13378343, -0.0403149575, 0.176398948, -0.00964029133, 0.123386756, -0.0300345421, -0.187632725, -0.0620219409, -0.188461006, -0.139842436, -0.100581177, 0.0265599042, -0.110380962, 0.191845462, 0.00141653419, -0.11816033, 0.208042368, 0.213605359, -0.129850671, -0.0933597088, 0.122598633, 0.00595799088, -0.018640548, 0.0378848463, 0.181395903, 0.173377052, 0.0876867622, 0.192007706, -0.209600434, -0.012859717, 0.00600273907, 0.127768829, -0.130987272, 0.134607062, 0.155363366, 0.0808825344, -0.0882706791, -0.076367721, -0.0793054253, -0.00586630404, 0.142082587, -0.206148043, 0.0407580584, -0.049249351, 0.0129451007, -0.116375081, 0.164335236, -0.105530523, 0.13251628, -0.0697510839, -0.0777705759, -0.117720746, 0.0540670604, 0.164986417, 0.103021309, 0.0867776424, -0.0438529849, -0.00377820432, 0.162118211, -0.128094852, -0.0133839697, -0.0300400108, 0.191699013, -0.114906885, -0.128097042, -0.125449896, 0.0672464222, 0.181721359, -0.0279202759, -0.0308043379, 0.012561053, -0.0228079483, 0.117388152, -0.0491030663, -0.152897894, -0.0109380297, -0.141598642, 0.12240307, -0.196314692, -0.139708713, 0.0969985127, -0.166283533, -0.261718482, -0.10953261, 0.0718631297, -0.213036582, -0.144475102, -0.00279817055, 0.0964064673, 0.0178181678, 0.110280976, -0.175311595, -0.251570255, 0.141161755, -0.188831225, -0.0564760268, -0.2272598, -0.152180851, 0.152426973, -0.00386719452, -0.0721517727, -0.012255799, -0.198725522, 0.105782107, 0.280836701, 0.0152221853, 0.275105059, -0.209379539, -0.224154338, -0.104977705, 0.0988008901, 0.0514465943, -0.0128156841, 0.157611817, 0.170334578, 0.0869703367, 0.285808533, -0.0728926361, -0.0931104496, 0.0235334337, -0.110741422, 0.125828728, -0.117568605, 0.155986264, 0.104506925, -0.0337914713, 0.0296717696, -0.235040098, -0.0135234362, -0.141636685, -0.100419141, -0.134680957, -0.186574012, -0.0766067058, 0.146882966, 0.154049531, -0.0364503711, 0.0356544703, 0.0556236356, 0.0494298339, -0.277094424, 0.073460117, -0.193379238, 0.134578362, -0.102159671, -0.239353925, -0.215223923, 0.194666088, -0.0964104012, 0.0814671591, 0.0992431194, 0.0468135215, -0.162915677, 0.162857607, 0.209440842, -0.187548369, -0.0020732081, -0.0355331898, 0.0981004983, -0.182766274, 0.0926911905, -0.0237608105, -0.102904551, 0.122693948, -0.236414105, -0.211930677, 0.115730271, 0.207284644, -0.0510552563, -0.157497108, -0.115445964, -0.173785508, -0.217097312, 0.103066951, 0.00525379414, 0.076337561, 0.12234731, -0.0626737922, -0.185681343, -0.0525672026, -0.0714665577, -0.215600729, 0.125220552, 0.0981240124, -0.178441167, 0.0892993957, 0.0875188187, 0.235276952, 0.0606884509, -0.0568252951, -0.242791384, -0.0947935879, 0.141819909, 0.204088584, 0.11860837, -0.0103346705, 0.143899903, -0.109179169, 0.103566274, 0.0646427423, -0.186479658, 0.200688288, 0.173446015, 0.191234097, 0.131643906, -0.0541896075, 0.17311503, -0.0397259891, 0.179010823, -0.160451055, -0.0738938302, 0.0460077673, -0.188182101, -0.167358577, 0.0334474444, 0.0105334073, -0.123536415, -0.0196802616, 0.15479432, -0.0144007057, 0.116810068, -0.208570942, 0.100825295, -0.19967401, -0.212417796, 0.0673297793, -0.215567753, 0.052130118, -0.151904643, 0.197143808, -0.0339394808, 0.206757233, -0.0573075712, 0.136985973, 0.108611509, -0.0870095193, -0.122860461, -0.1796031, -0.0982395262, -0.101981603, -0.107995287, 0.140654042, 0.170272157, -0.124455385, 0.119262144, 0.163930461, -0.185422182, -0.21241951, -0.121740013, -0.172264829, 0.0637018234, 0.051629886, -0.14822641, -0.112850063, 0.0174066424, -0.0829333961, 0.0977343246, -0.071891427, 0.0561515987, 0.109630719, 0.0105861574, -0.0270061102, -0.190160096, -0.119579576, 0.197185382, -0.0970397443, 0.0522243232, 0.000522117305, 0.0153891267, 0.146401003, 0.159108639, 0.25341928, 0.00318193459, 0.0668381304, 0.0247753933, -0.115337625, 0.0172942206, 0.0831532627, -0.0902798697, -0.105036713, -0.213386223, -0.121249683, 0.0464711972, -0.141757503, -0.113185756, 0.193994313, -0.187768489, -0.15975529, 0.0177620109, 0.0166279227, -0.193038374, -0.0627801642, 0.0224070493, 0.105940476, -0.137638792, -0.11995957, 0.0115957642, -0.128734171, 0.138942927, -0.108310811, 0.0426762067, -0.234138444, 0.0704599395, 0.113127954, 0.180509791, 0.169870883, 0.0833347514, 0.112489417, 0.11732848, -0.0221389327, -0.110925816, 0.117433928, -0.214904755, 0.054917559, -0.0237672813, 0.148916826, -0.017192632, 0.0826454312, 0.164108485, -0.0137663055, -0.0730242953, 0.234863907, -0.178744644, 0.0621348992, -0.00839559734, -0.10974963, -0.0248806775, 0.055587817, -0.0795170292, 0.18179898, -0.149376124, 0.0317146517, -0.0143466592, -0.0674705505, 0.17889294, 0.0754329786, -0.150365472, 0.0464622527, -0.00969791599, -0.200375721, 0.0205095354, 0.154160127, -0.00569080515, 0.155038372, -0.0677913055, -0.147895366, 0.0321660787, -0.056184493, 0.0394759253, -0.157382205, 0.233074352, -0.0469223112, 0.116115957, -0.203592524, -0.123089239, -0.164869681, 0.0379196517, 0.0770090148, 0.0427877568, -0.169947818, 0.0919543505, -0.0403930247, 0.175416812, 0.21293062, 0.210629076, -0.111974031, -0.14331843, 0.0128842229, 0.0350685567, 0.0866905451, 0.13432996, -0.202785864, 0.0997599959, 0.207019001, 0.138129339, 0.0494085439, -0.108375512, -0.127402216, 0.0275171027, -0.0740583614, -0.00576845882, 0.193134576, -0.0666644946, 0.0633924752, -0.089058876, -0.0918698311, 0.0843076035, 0.202469081, 0.0892445296, -0.1374605, 0.0150794983, 0.0531005375, 0.161458567, 0.210192963, 0.04205136, 0.107358694, -0.0251380932, 0.0682467371, 0.186786473, 0.0294182803, 0.0918548927, -0.197670788, -0.144377872, -0.191045746, -0.20302172, -0.0703191012, 0.26318568, 0.183188379, -0.206453308, 0.217197284, 0.148158118, 0.0516163856, -0.0405543372, 0.0482969098, -0.0797786266, 0.0162452161, -0.142858282, -0.0700473189, -0.165941894, 0.0412169918, -0.200823486, -0.21580334, 0.0719728321, 0.0922091603, 0.149025053, -0.023213055, 0.265344322, -0.150436535, -0.021344753, -0.140235752, -0.255674452, 0.15332745, -0.00951609015, 0.165915266, 0.0167089067, 0.124824308, 0.0771664828, -0.253194153, 0.0453373007, -0.0910207182, 0.0636530071, -0.19644013, -0.231708229, 0.178851888, 0.18904604, 0.0673967227, -0.253504723, -0.004631266, 0.0158821791, -0.0782575011, 0.112024978, 0.0643248707, 0.0634058863, 0.00650183856, 0.0145138055, 0.0211943984, -0.186126992, 0.153037265, -0.0982570276, 0.117266491, -0.0641367286, 0.0506336838, 0.177407131, 0.027125746, 0.08834593, -0.170427591, -0.156710893, -0.180125281, 0.18578954, 0.132006899, 0.0475857705, 0.0842403024, -0.0162469745, 0.103354886, 0.208519891, 0.194094405, -0.0861671567, 0.138932332, 0.201304033, -0.193600982, 0.175816432, 0.107227907, 0.169770226, 0.0631686598, 0.0528858155, -0.0414999276, -0.104278192, -0.17777279, 0.107138261, -0.0946334153, 0.0493052155, 0.195973918, -0.0339171737, 0.167163864, 0.062439546, 0.191270575, -0.204546601, 0.204385087, -0.0609797537, 0.102811083, -0.0426427275, -0.144036323, -0.215613484, -0.149330556, 0.186492875, -0.112123109, -0.129927844, -0.153668568, 0.0724345893, -0.147795394, 0.195619091, -0.168710485, -0.0126553029, -0.0127404332, -0.116737291, 0.168202505, -0.139484406, 0.0554534048, 0.0361851305, -0.113191009, -0.174208596, 0.0114807189, -0.195487082, 0.134786084, 0.144725397, 0.207942024, -0.0374336243, -0.0180579275, 0.1983376, -0.0727393627, 0.0687315911, -0.0218542069, 0.0489843339, 0.160994157, 0.0465723425, -0.0552227646, -0.160425812, 0.118589506, -0.173039734, 0.094873175, 0.0973959714, -0.0334962308, 0.131362393, 0.192723766, -0.085611105, 0.186923936, 0.173444375, 0.195655927, 0.0500997752, -0.0955151692, 0.0853087157, 0.109827921, -0.0743474066, -0.135200426, -0.0115245879, -0.024191156, -0.0558120608, -0.160451472, 0.0763798505, -0.16293782, -0.1017408, -0.15939261, 0.0827288479, -0.215683803, -0.0368343294, 0.0422128886, -0.176073387, -0.105860367, 0.0477225035, -0.115710489, -0.193383917, -0.188803807, -0.170165524, 0.0757941753, 0.16839464, 0.0277366079, -0.123203889, 0.094133839, 0.195007026, -0.202828094, -0.105727762, 0.0652255863, -0.166010231, -0.126647398, -0.0466658585, -0.120006435, 0.0939842612, -0.0244721789, -0.194358811, -0.0313170701, 0.109878041, 0.194994539, -0.148321584, -0.154995516, -0.0752039999, -0.0561695024, -0.0345148742, 0.0120506845, -0.145251185, 0.276574999, -0.183512345, 0.246295869, 0.175020978, -0.134096593, -0.171224758, -0.178246081, -0.0637267604, 0.0260362774, -0.0426347815, -0.0999041423, -0.133127928, -0.217847079, -0.195832476, -0.108974583, -0.00344945025, 0.247975796, -0.0544710569, 0.0776171461, -0.0458349697, -0.232248828, 0.0165108331, -0.16456145, -0.118792772, 0.135833904, 0.191254571, 0.152048305, -0.0461367741, 0.116522327, 0.00936230551, 0.0552281439, -0.00196163752, 0.229142398, -0.142573804, -0.0892553627, -0.120750993, 0.256958574, 0.0426204354, 0.0873946771, -0.226227716, 0.141678169, -0.042470932, 0.124623254, -0.179483652, -0.116647683, -0.116587028, 0.103890166, 0.123260602, 0.0605796427, -0.0168686211, -0.00929376483, -0.0128240585, 0.172887877, -0.0799608827, -0.0303717256, -0.127870053, 0.17608051, -0.0424753278, -0.0972225741, 0.0391885191, 0.200019762, -0.0154580772, -0.186458692, 0.134563908, -0.0995464176, 0.0737005621, 0.176864192, 0.0450127572, -0.188842878, 0.0309933126, 0.0700256974, -0.0154144019, -0.0797051638, 0.187247232, -0.0477865189, -0.0276180953, 0.180766746, -0.199228138, 0.207444504, -0.16353789, 0.156251594, 0.165612713, 0.11059694, 0.209873334, -0.140326887, 0.175071821, 0.0395414978, 0.156043813, 0.0787585527, 0.199952558, -0.0327560008, 0.0251382589, -0.199105844, 0.0476279408, -0.0291632563, 0.0443746597, 0.173739001, 0.00965835154, -0.117652602, 0.0828595608, -0.164778814, 0.156857237, -0.130015075, -0.107045695, -0.222709522, -0.0534569211, -0.146377668, 0.143743783, -0.223435938, 0.0202661306, 0.0298079774, 0.130296096, -0.169427738, 0.0867685452, -0.189785749, -0.214855, 0.138201609, 0.0175307598, -0.00683422387, -0.0721608624, -0.148823351, 0.0987624824, 0.163937375, -0.221082836, 0.097356841, -0.10563866, -0.174024582, 0.231104016, -0.167891935, -0.0109430226, -0.0339421071, -0.015225037, -0.0966599807, -0.0566251948, -0.038483344, -0.0632045045, -0.173830792, 0.234540999, -0.0372984409, -0.11684528, -0.0237086806, 0.177134946, -0.135995328, 0.143075436, 0.0284443703, 0.0957668871, -0.203221127, -0.138940528, -0.170615286, -0.04803662, -0.0227327403, 0.156518131, -0.120296806, 0.116717979, -0.0278942138, -0.180543825, -0.120960377, 0.0104260044, -0.125010282, 0.105188407, -0.0110195624, 0.0892315656, -0.200755909, 0.205126464, 0.168077156, -0.118845731, -0.142220959, -0.0858293474, 0.0769720748, 0.00681600207, -0.0523019433, -0.109635837, -0.0064796377, 0.0102793276, -0.130109623, 0.150559291, 0.0784872174, -0.0432755277, 0.188085303, 0.00808112323, -0.181910425, 0.0972780362, 0.138851807, -0.165652379, -0.167549655, 0.123791538, -0.212279394, 0.103910975, -0.124968246, -0.0679621696, -0.150251463, -0.0412153937, 0.18648304, 0.171684593, 0.00163652177, -0.138664946, -0.0801473856, 0.176220953, -0.181696028, -0.00872888416, 0.181269154, 0.0954500809, 0.0857712477, -0.137488693, -0.0543198027, -0.168690518, -0.210396335, -0.211841181, 0.111533284, 0.0498711616, 0.131123632, 0.171156824, 0.0636221096, 0.0163842924, 0.00664749416, -0.193607077, 0.104148954, 0.0818801969, -0.126201361, 0.107612975, 0.109677412, -0.132316753, -0.0396888182, -0.00945395418, 0.0487647355, 0.0377194248, 0.178009942, -0.135111406, 0.137946114, -0.0810011625, -0.0691107288, -0.182944283, -0.0679595321, 0.0203998834, 0.174737379, 0.0201928318, 0.0889042467, 0.0805583745, -0.204121158, 0.00436645746, 0.0794607848, 0.0822678357, 0.00139918923, -0.0264118016, 0.0835606307, -0.00963528454, -0.0870883018, -0.12715739, 0.145659909, 0.0546541363, 0.187282696, 0.0855048746, -0.0967017934, 0.0764478296, -0.208491907, -0.0981765538, -0.017935276, 0.127355561, -0.124414347, 0.0346565694, -0.108974963, -0.0984654129, 0.125999585, 0.0118691027, 0.0898878127, -0.0464704335, -0.00716736913, -0.0696949661, -0.00315192342, -0.172756493, -0.034152925, 0.0687169284, -0.0139536262, 0.0157241225, 0.0378018171, -0.0701506585, -0.00593361259, 0.16699715, -0.0711576492, -0.043457225, 0.127052858, -0.0215502083, 0.177768037, -0.0212931484, 0.12964575, -0.196589366, 0.0531259924, 0.023148343, 0.15855442, -0.0950687155, -0.0336764306, -0.0928969979, 0.197106078, -0.0703088194, -0.0125174373, 0.104199722, 0.0937243253, -0.0498488285, -0.0790696591, 0.0754235014, 0.159118399, 0.175383911, 0.00834533945, -0.132660657, -0.115502544, -0.0156698935, -0.142873257, -0.172217071, 0.00926896464, -0.0980520546, -0.186849445, 0.104777038, 0.141713575, -0.116373293, -0.177874327, -0.0812455565, -0.180731073, 0.157215104, -0.0100824358, 0.13991484, -0.165303022, 0.129494235, 0.102651075, 0.0760747492, 0.0534787029, -0.201117173, -0.148061618, 0.158403665, 0.170118049, -0.184529886, 0.00612172484, 0.18630074, 0.0668295771, 0.203014389, 0.0470853746, 0.120209262, -0.0326153599, 0.178558037, 0.130264938, -0.158517003, -0.236181453, -0.077458322, 0.0907330364, 0.0622364357, 0.118951038, 0.0970379859, 0.157590434, 0.0286808833, -0.103834197, 0.0967250317, 0.052686438, 0.0817455575, 0.121504307, -0.154424161, -0.16611585, -0.130731776, 0.194687054, 0.186306313, 0.00081812439, 0.0815480202];
    bias_1 : ARRAY[0..63] OF REAL := [-0.00991463661, -0.000165412683, 0.0380159281, -0.0313414298, -0.00776600698, 0, 0.0327618271, 0, 0.0053440691, -0.012447658, -0.00528640207, 0, 0.00980756432, 0.0239994954, 0, -0.00600226782, -0.0427969247, -0.0124991806, 0.0102020688, 0.0347996801, -0.0137349106, -0.00922023784, 0.060131371, -0.043544095, -0.0354361534, -0.00553967617, -0.0374039412, -0.030632956, -0.00583763421, 0.00989670772, -0.00822056364, 0.0306522157, 0, 0.0557479262, 0, 0, -0.00697317952, 0.0160537008, 0.0252484679, -0.0129459258, -0.0292139072, -0.038203638, 0.0335591063, -0.0462469868, 0.0442246161, 0.0594434552, 0.0479242764, 0.0381261297, -0.0195034202, 0, -0.00470581418, -0.00563494209, -0.0306187645, -0.0391318202, 0.0379941873, 0.0250570383, -0.0389060415, -0.00584178604, 0, 0.00260822545, -0.0485509746, -0.0251302961, -0.00867041945, 0.0280207619];

    weights_2 : ARRAY[0..4095] OF REAL := [-0.141680449, 0.288066953, -0.150528222, 0.0983807966, 0.0682033002, -0.0383133292, -0.0808929056, 0.143694162, -0.143791497, 0.173556536, 0.0320169441, -0.121532038, 0.0184226483, -0.0103868982, -0.0746624023, -0.135166839, 0.113171645, -0.126689032, -0.0239767376, 0.0532080457, -0.10377644, 0.104337208, 0.0625005439, -0.119132705, 0.202529803, -0.086342141, -0.205905676, -0.150743365, 0.0873293057, 2.73770947e-05, 0.064553991, -0.0785556436, -0.157094628, 0.00396119431, 0.0939819738, -0.0202242639, -0.150879264, 0.125680909, -0.0767421126, 0.107631303, 0.0793541521, 0.0918624699, -0.0373493209, -0.227653801, 0.16160652, -0.210584804, -0.000720652053, -0.13250798, -0.103983767, -0.123876065, 0.029696513, 0.177454278, -0.053838402, -0.105550319, 0.115103669, -0.0959799588, 0.18597813, 0.231739312, 0.135426775, -0.046401687, -0.100035861, 0.0408016182, 0.0825353414, 0.136485547, 0.00270199776, 0.0867017061, 0.195101574, 0.126894072, -0.132388622, -0.0208239406, 0.00692871585, 0.128494516, -0.13354221, -0.0511906333, 0.0144319832, -0.171571314, -0.125738502, 0.13592577, -0.137273088, 0.1709162, 0.0410082564, -0.183967724, 0.0714212805, -0.0134086907, -0.0914759263, -0.111280508, 0.182648227, -0.0738228038, 0.0616786629, -0.21075432, 0.203339309, 0.0925859734, 0.115103915, 0.0693822652, -0.188044399, -0.108215593, 0.164470464, 0.153212592, 0.0917293802, -0.179572374, -0.143311441, 0.115444198, 0.0727809519, -0.00865674019, 0.127544686, -0.0877099037, 0.103159383, -0.078883104, -0.100927807, -0.0344764031, -0.12042328, 0.0344114751, 0.131927297, -0.146454126, 0.0510100611, -0.0590627939, -0.0506405383, 0.0810800865, -0.090818353, 0.0528705269, -0.201525137, -0.0838072225, 0.110697366, 0.0740895495, 0.172959939, 0.189559668, -0.065729633, -0.0720220059, 0.105840042, -0.058448758, -0.107932165, 0.216511503, 0.00461578369, -0.107524514, 0.058490552, -0.175286993, 0.0249149054, 0.0852858871, -0.157516927, -0.0535053015, -0.0676146448, 0.0599285662, -0.0855296031, 0.140303031, 0.149562418, -0.0901874602, -0.0450080633, 0.0728893131, 0.00284661353, -0.0671322271, -0.105737545, -0.0900957286, -0.198729545, 0.162473515, 0.147394195, 0.145424545, -0.0517513901, -0.0669851601, -0.164583072, 0.110631853, -0.215715826, -0.170075879, 0.0506092906, 0.00326168933, -0.0199967101, -0.0183630344, -0.0711533353, -0.148096681, 0.114399835, 0.0869136602, -0.115128055, 0.156051964, 0.14734675, -0.148528323, 0.104175396, 0.282105029, -0.235148892, -0.208776742, -0.088167496, 0.198368117, -0.205772802, 0.00897102989, 0.0128333028, -0.0552920029, -0.166966945, 0.147610545, 0.0774816051, 0.0655531734, 0.146716073, -0.00372734619, -0.214626014, -0.0576679409, 0.00339318812, -0.0645904765, 0.129015684, 0.0367895626, 0.00563158561, -0.150251627, 0.14424403, 0.219185576, -0.015582785, -0.0557845123, 0.229870901, -0.136385068, 0.193651333, 0.0781679228, 0.10057772, 0.0421372652, -0.078148827, 0.111039303, -0.0640359819, 0.213664457, 0.239976257, 0.134989008, -0.121206947, 0.158595756, -0.170423076, -0.138676971, -0.0604084283, 0.129199952, 0.163071141, -0.221609473, -0.0275269188, 0.186735034, 0.13408266, 0.0231132358, 0.196531892, 0.0723142847, -0.184686705, -0.0832601115, 0.130843252, -0.0489593074, 0.182337478, -0.0457641892, -0.00743399095, -0.126927346, 0.0406110212, 0.0973830223, 0.188993767, -0.0883924365, 0.263101488, -0.0826768279, 0.15883705, 0.172388598, 0.123626038, 0.10255266, -0.252580434, 0.211067945, -0.0147316307, 0.00241988176, 0.156785056, -0.112871908, 0.0347109661, 0.0922119021, 0.00649048388, 0.153683811, 0.138896421, 0.0972352177, -0.208112851, -0.202854082, 0.0617144667, 0.0563855022, -0.0516398437, -0.0742861032, 0.0109137893, -0.117585734, -0.0220603198, -0.0585992336, -0.0475497693, -0.0259862747, 0.119525358, 0.189453453, 0.172370642, -0.0726865008, -0.0956337899, 0.0137653798, -0.150756568, 0.118895762, -0.083567664, -0.165870577, 0.130793914, -0.133739084, 0.198176801, 0.184771329, -0.209565952, -0.183116794, -0.0640594736, -0.203715086, 0.0997374058, -0.070866093, -0.171968624, -0.122551396, 0.0937422961, 0.19882901, 0.120841727, -0.00538546452, 0.199771121, 0.121376611, 0.141540334, 0.159105301, -0.0297715347, -0.196540907, -0.124991439, -0.145521253, 0.205668867, -0.0768398345, -0.035737481, -0.0238609333, -0.124907829, -0.0484834574, 0.124906845, 0.124305926, -0.0377987772, -0.191355884, -0.159768522, 0.183061063, 0.184881866, -0.212566867, -0.0531422645, 0.0976230353, 0.00577385724, 0.130427197, 0.211715534, -0.0860495567, 0.0888584703, 0.121544942, -0.180683181, -0.0218638033, -0.0905238539, 0.0180363953, -0.02386415, -0.13335371, -0.00121800601, -0.094210498, 0.112201318, -0.216103971, -0.0530306548, -0.158522308, 0.152102396, -0.15442571, -0.134984136, -0.0138640255, 0.0654296428, -0.158441991, -0.134703487, 0.190590188, -0.176293343, -0.178531021, 0.0348580927, -0.00753350556, -0.213596776, 0.109840617, -0.103785381, -0.0846005082, -0.082864821, 0.108093217, 0.132263497, -0.156487495, 0.149631396, -0.0340299606, -0.0305996239, 0.107479975, 0.0321970284, 0.0810965151, -0.169963852, -0.0118091106, 0.173262879, 0.134186372, -0.20041047, -0.000686064363, -0.0538731366, -0.0124969929, 0.0516002327, 0.0954418629, 0.0455744714, 0.0564913601, 0.133059844, 0.110250726, 0.180289343, -0.000993043184, 0.186119303, -0.0665116161, -0.0792722255, 0.202967927, 0.205843329, 0.21862179, 0.0488890447, 0.0133959213, -0.00834459066, 0.00461511314, 0.0836300105, -0.121354386, 0.117611662, -0.234934494, 0.0287881922, -0.0978208929, 0.136924744, 0.0765881464, 0.148768306, -0.168677807, 0.0451220796, -0.0645759478, 0.182842463, 0.139968216, 0.0730862394, 0.0406570174, 0.0715097487, -0.159143537, -0.122275874, 0.147242293, -0.146196708, 0.0239535533, 0.10290198, 0.0115962736, -0.0944432169, -0.0756312534, 0.0423654877, -0.168181121, -0.0449682809, -0.0617624037, 0.152064502, -0.0231318604, -0.0633203983, -0.00436079642, -0.110454418, -0.246325403, 0.188381672, 0.122344673, 0.123941295, 0.201515913, 0.24498114, 0.182052374, -0.163516134, -0.156467408, -0.00582023244, -0.112946808, -0.127423167, -0.0515909754, 0.155103877, -0.173389852, -0.199556112, 0.115317613, -0.162211671, -0.191533402, -0.0836257115, -0.0725069493, 0.06501095, 0.035802599, -0.176167637, -0.0298467577, 0.155019239, 0.169515267, -0.000437632203, -0.0261323899, 0.199166045, 0.172561631, -0.193425417, 0.175140068, -0.0974695757, -0.142100155, 0.194233581, -0.0656768829, -0.120199233, -0.162119597, 0.169042096, -0.214600414, 0.0662081391, 0.0520145446, 0.107069895, 0.175651714, 0.131947085, 0.143850192, -0.00955465436, 0.0627427548, 0.210242525, 0.0844678432, -0.129487574, -0.0942333117, -0.0245972425, -0.090298906, -0.0466166288, -0.107186824, 0.111454025, -0.137471825, 0.136128113, -0.0861810446, -0.186852902, -0.0583910942, -0.0535676479, 0.0353205353, 0.0871732086, -0.146667257, -0.121421315, -0.143794656, 0.147011802, 0.170059487, 0.0102381408, 0.153043762, -0.00729104877, 0.0746920556, -0.0543518513, -0.0595977008, -0.0225165188, 0.0500841886, -0.182219625, 0.0947217196, -0.205081433, 0.12140505, -0.201528907, -0.0524655879, 0.155590281, -0.129846334, 0.0906220675, 0.151344299, 0.186176911, 0.0421557426, -0.207316592, -0.131616503, 0.133107722, -0.160803005, 0.143145278, -0.161467314, -0.0657405034, 0.135806978, 0.166633621, -0.200071856, -0.207391843, -0.215113148, 0.148792446, -0.0100589618, 0.0714959651, -0.0805551559, -0.0614150316, -0.174764574, 0.207058311, 0.122847259, -0.196977898, -0.1559522, 0.0978694558, -0.185000882, -0.140967488, -0.16737549, -0.106714033, 0.164967701, 0.0964245871, 0.140171438, 0.207501814, -0.0379861556, -0.0579505898, 0.225760758, 0.111228764, -0.146074057, 0.0667390376, -0.169152468, 0.938151181, 0.17469056, -0.175612152, -0.123244651, -0.126487702, -0.0329091251, 0.138695627, 0.0742424577, 0.098279722, 0.119007275, -0.172866449, 0.0933431759, 0.0521263108, -0.131282881, 0.0761865526, -0.0664989054, 0.164532125, 0.0566500686, 0.200022459, -0.0600383841, 0.182312235, 0.194255427, -0.0288380273, -0.122255489, -0.0914943814, -0.0893590152, -0.0746954307, 0.146213099, 0.184557945, -0.118034557, -0.174534202, 0.0035078912, -0.0207415409, 0.105583005, 0.0245418437, 0.184224337, -0.0410954989, 0.113560788, -0.0217513908, 0.0455570407, 0.0366436318, -0.159584582, 0.0670233443, 0.21683304, -0.128995791, 0.275691748, -0.0195934419, 0.177997693, -0.1972785, -0.0668776929, -0.216343522, 0.163236275, 0.205884218, 0.216626123, 0.147940427, -0.0883644, 0.092634283, 0.207626119, 0.171906605, -0.167044088, 0.204324439, -0.109410673, 0.0193916559, -0.119002052, 0.0720684603, 0.141300142, -0.088518776, 0.0176712964, 0.161592081, 0.126937598, -0.0751166046, -0.133596882, -0.115226425, 0.24855116, 0.122299738, -0.095500432, -0.119029626, 0.152431637, 0.00319294631, 0.21932444, -0.0965302214, 0.134576872, -0.015701618, -0.0857832581, -0.216072649, -0.137355849, -0.196437761, -0.126480833, 0.0231357962, -0.134333387, 0.171409652, -0.113697752, 0.0360458046, 0.163777098, -0.0132845491, -0.153503746, -0.213196114, 0.0580244511, 0.152173683, 0.0331603885, 0.211798117, -0.199593693, 0.129404142, 0.113514826, 0.0272548497, -0.214540333, -0.193730131, 0.215466887, 0.0018462775, 0.013003692, 0.195035413, -0.0590138286, 0.0399461836, 0.0308904201, 0.179027125, 0.0488234572, 0.0415520221, 0.137228593, 0.200982258, -0.156045571, -0.105913378, 0.133550122, 0.0291233379, -0.081467703, -0.145602509, 0.171516255, 0.0566335171, -0.00745478272, -0.167673349, -0.118719235, -0.00841763616, -0.167444021, 0.0689675286, -0.200617492, -0.121176332, 0.0399130136, -0.194600999, -0.107290849, 0.201394126, -0.0595335364, 0.197396234, -0.0294916183, -0.0975661054, -0.0199405309, -0.0464265756, 0.0777761638, -0.184141561, -0.0692353547, 0.203581437, -0.0510522276, 0.00841990113, -0.0510387868, -0.209235489, -0.0786187798, 0.0127682984, -0.0585706383, -0.149550289, 0.0406086594, -0.15494749, -0.0766567886, 0.192089304, -0.174240753, 0.168413922, -0.184974745, 0.129347548, -0.0480398685, 0.102323428, -0.00398623943, -0.0793017, 0.186511293, -0.01932621, 0.140939757, -0.008235991, 0.135236308, 0.0234718472, -0.0376885831, 0.0408930033, -0.0838549286, 0.105532184, -0.169196993, 0.00895322859, -0.0224669725, 0.214271948, 0.187380776, -0.168133691, -0.171357155, -0.0451917201, -0.090357855, 0.126548275, 0.102986887, -0.133371353, -0.0108436346, -0.0374744087, -0.17570509, -0.132929906, 0.00220645964, 0.127038345, 0.0997535139, 0.210657284, -0.137902528, -0.125172943, -0.21302484, 0.10058029, -0.0661100745, -0.00623327494, 0.0631183833, -0.103329279, -0.185445309, -0.0871112198, 0.0991731733, -0.194505647, -0.200181127, -0.0255591124, -0.205262512, -0.204970762, 0.0392911546, -0.20052886, -0.0514694117, 0.0394407958, 0.0124119818, 0.130332097, -0.101388983, 0.137814477, 0.0253826454, 0.190587938, -0.161746755, -0.198715627, -0.077888988, -0.0540392175, -0.096387893, 0.00343954773, 0.113467187, 0.166445121, 0.0665265769, 0.115969144, 0.16848965, -0.114840552, 0.164357632, -0.0157545805, 0.191388026, -0.175001413, -0.131909996, -0.0113435686, 0.147116452, -0.0923970491, -0.0562144518, -0.176853389, 0.0598261133, 0.190945908, -0.0372008011, -0.0430109315, 0.11451865, 0.0371341594, -0.0761518031, 0.110607252, 0.00426071882, -0.146474242, 0.0800529569, -0.11710421, 0.0366946682, 0.269265682, 0.191883326, -0.0611798316, 0.00541722775, 0.232036233, -0.202542618, -0.14030695, -0.0281257648, 0.230240002, 0.0162147321, -0.164047837, -0.124143533, -0.121437646, -0.17262505, -0.0583858602, -0.0723832101, -0.19505994, 0.0283917375, -0.131140262, 0.0902625024, -0.115805745, -0.117771566, -0.116753951, -0.0244481117, 0.154554754, 0.0925760716, -0.177714929, -0.0415367521, 0.0639798269, -0.128405958, 0.0617773086, 0.12867713, -0.220567599, 0.155001327, -0.164517075, -0.10119269, -0.0264345706, 0.193819627, 0.00867548306, -0.131352246, 0.168402314, -0.0690761581, 0.0819703862, -0.124435671, 0.12688598, 0.113567822, 0.0819837376, 0.236767009, -0.196865633, -0.0627399534, -0.167267427, 0.0447263867, 0.211083233, 0.127811357, 0.144808367, -0.108109578, -0.0729895085, 0.103431262, -0.130963951, -0.0642541945, 0.0399866477, -0.0517324097, 0.106077358, 0.0571983159, -0.137635872, 0.172099277, 0.171573251, 0.0966628045, 0.0747942552, 0.0563847944, -0.0897115842, -0.182717025, 0.0567689948, -0.0702779293, -0.0933412313, 0.165129632, -0.0129972473, -0.0846574679, 0.128517389, 0.12487001, 0.170890465, 0.18792893, 0.111724451, 0.177234873, 0.160684839, 0.0530777425, -0.0586484224, -0.160080284, -0.144362509, -0.159860179, -0.181875899, 0.154358193, -0.0374765694, -0.083326295, 0.181780145, -0.121391997, -0.0691839457, -0.0742421448, 0.0691870898, 0.14754726, -0.069750309, 0.0740958601, 0.198498741, -0.154731348, 0.0730743259, -0.00451502204, 0.0863774866, -0.092950426, 0.131180331, -0.18926172, 0.148594961, 0.0665854961, -0.0706014037, -0.0448699296, -0.0694603622, 0.0639980286, 0.0166171342, 0.196238205, 0.016624555, 0.0550233275, -0.180780441, -0.161480352, 0.0111390948, -0.0118472576, -0.0242867023, 0.0894839317, -0.214834765, 0.165922478, -0.146362454, -0.205421194, -0.146823198, 0.0966032892, 0.148615941, -0.0852327496, 0.163918838, 0.102714762, -0.208166033, 0.0172590613, -0.0552005172, 0.0110155195, 0.179708347, 0.0191160589, -0.133684993, -0.0525586009, 0.205576107, 0.210995749, -0.138825268, -0.142582893, -0.141632929, 0.0855522454, 0.198174328, 0.00804278255, -0.0469306856, 0.0574738979, -0.144030869, -0.165960878, -0.108321778, -0.197332725, -0.0156382918, 0.0518989488, 0.0718663186, -0.0900121629, -0.0854760781, -0.216951966, 0.180414304, 0.0896183103, -0.0315984115, -0.038237486, 0.16515182, -0.0816439539, -0.0227444768, -0.0454315543, -0.185322598, 0.0210614055, -0.194109529, 0.0599969067, 0.0527030006, 0.0741187185, 0.156095579, -0.0249356292, -0.164651155, 0.123715535, 0.172677234, -0.0501076728, 0.0449018963, -0.0228640102, -0.0200645179, -0.084004961, 0.0933688506, -0.12003617, 0.146246135, 0.114758648, 0.0661290213, 0.126682028, 0.161090702, 0.140608266, -0.148477748, -0.0640800446, 0.133195326, -0.0674081072, -0.181248829, -0.0289781466, -0.0194690824, -0.0494243838, 0.106817186, 0.195835143, -0.0803123191, 0.161425516, -0.0493547022, -0.05296278, -0.196740344, -0.17108798, -0.0269036777, -0.257117361, 0.0609735921, 0.126235262, 0.234910175, 0.298613906, 0.110691503, 0.163770065, 0.164086029, -0.102102607, 0.269784272, 0.298873127, -0.141947195, 0.00401810464, 0.160247535, 0.199671581, 0.102458611, -0.171934664, 0.211893931, -0.109412298, 0.0464521386, 0.174394637, 0.0244902223, -0.0639190525, -0.0315829515, -0.0628100634, -0.145441294, -0.248165399, -0.096565783, 0.0521190837, 0.171565145, -0.0265039522, 0.113324709, -0.0879507959, -0.022442922, -0.175112098, 0.194249406, 0.0624903068, -0.174791113, 0.0232726112, -0.254210442, -0.126247719, 0.245405003, 0.154142827, -0.183761641, 0.124047622, 0.143147632, -0.11987894, 0.0924994051, 0.238024503, -0.0995406434, 0.127400458, -0.118362844, 0.0286737774, 0.0726793855, 0.0532515496, -0.00276745413, 0.147954509, 0.175074711, 0.263851762, 0.0354693085, -0.0399195738, -0.0167579949, -0.0360376686, 0.119187571, -0.175929293, 0.179050192, -0.209990561, 0.0303346924, -0.0304141119, -0.168580458, 0.0159338806, -0.143411383, -0.14976643, 0.0935455635, -0.0950493068, 0.0929078311, 0.0551954135, 0.0518541336, 0.176312774, -0.183571264, -0.102172591, 0.174365237, -0.10537722, -0.041147884, 0.0739963651, -0.111693986, -0.0890176594, 0.0285699144, -0.157434717, -0.14237228, -0.00719396165, 0.0457479246, -0.146615341, -0.07867226, 0.00846140739, -0.130273566, -0.117995292, 0.0493791625, 0.183448762, 0.148034781, -0.191158175, 0.15299876, -0.0805099756, -0.0233456288, -0.168751732, 0.00436502555, 0.139199287, 0.193048775, -0.143146724, -0.197523668, 0.112838462, 0.0882283896, -0.176614121, 0.0627285391, 0.115050167, -0.203107342, -0.130106881, -0.0552822948, -0.10732834, -0.131432489, 0.0808235332, 0.217252836, 0.0871307775, -0.0174604356, -0.165878817, -0.172403678, 0.254087269, -0.162096322, 0.323802054, -0.012599051, 0.151775375, 0.153595924, 0.00913618691, -0.182565987, 0.114645109, 0.0815113634, 0.121357247, 0.126867056, 0.0927122906, -0.136515841, 0.106271967, 0.209716767, -0.152262896, -0.0599813312, -0.0153267533, 0.0652863383, 0.219464377, 0.196837217, -0.223917902, -0.143790111, 0.138385013, 0.113471806, 0.367199123, -0.137293875, -0.0288341846, -0.0667795986, 0.038723208, 0.102534734, -0.138440862, -0.0140577843, -0.0820909142, 0.329797894, 0.0938638672, 0.0398048386, -0.20963259, 0.154240653, -0.0378240161, 0.134357706, -0.0533082113, -0.0598759018, 0.0404425971, 0.21940358, -0.00829724967, -0.120814763, 0.0788223594, 0.11621587, -0.20682922, 0.00859716535, -0.00990748219, 0.0331411287, 0.114033349, -0.151647523, -0.158313036, 0.0926335678, 0.0706593469, 0.351727486, 0.166647702, -0.0461413115, 0.216942608, -0.138307035, 0.144426495, -0.169870242, 0.200646102, -0.16545783, 0.181138262, 0.11609225, 0.077415742, -0.182514325, -0.15969798, -0.21806176, -0.160868764, 0.104007304, -0.160312831, 0.0297145694, 0.0499397293, 0.0594710223, -0.0964953378, -0.177800402, -0.0670034215, -0.19343999, 0.180497482, -0.0837211534, -0.128186598, -0.13259843, -0.089160189, 0.0347441472, 0.128377378, 0.105255894, 0.11304494, -0.158335477, -0.183520451, -0.132612199, 0.195470482, 0.171718106, -0.21191743, 0.176613376, -0.0911389291, 0.0547690429, -0.122613512, 0.0449908227, -0.0874788165, -0.0113770878, -0.102273077, 0.125744522, 0.0171495155, 0.103814244, 0.185875043, -0.0773060992, -0.207971171, 0.0723132193, -0.0591497123, -0.174698785, -0.0662334561, 0.0624778345, 0.181660056, 0.0352354199, -0.144429192, -0.0237713046, 0.1413863, -0.055128105, 0.107294582, -0.0923522636, 0.10639482, 0.0696970969, -0.104372099, 0.0329963788, -0.142583638, 0.197051004, 0.039161697, -0.0938943475, -0.0997598544, -0.0650602877, -0.0785568804, -0.0371245071, -0.13516289, 0.00734080002, 0.0694661215, 0.0717197061, -0.038889166, -0.0539452471, 0.213663176, -0.0399716944, 0.015419662, 0.0576197021, -0.211071417, -0.00350436778, 0.15874508, -0.0291592199, -0.0852676928, -0.186650351, -0.143953145, 0.160483733, 0.23401615, -0.174104869, -0.0815619752, 0.178066641, 0.206289992, -0.13791053, -0.162200421, -0.111578882, -0.0799070597, 0.137941718, -0.109797254, -0.0264309049, -0.0568498187, 0.0664690062, 0.0718042403, 0.0974657089, 0.0933575481, -0.0164596867, 0.210323125, -0.142812029, -0.149296373, -0.180004731, -0.0265571047, 0.128158346, 0.0553876162, -0.122902334, -0.0440571681, -0.112295315, -0.138417289, 0.039254874, -0.193141863, 0.0195326358, -0.201830551, 0.150758162, 0.115440972, 0.202520981, 0.106997013, 0.0990103036, -0.129501849, 0.0595938414, 0.090642944, -0.112931691, 0.0857426375, -0.152478904, 0.144109204, 0.0355113298, -0.107244223, -0.0304977745, 0.113781944, 0.12506713, -0.207027107, -0.182988301, -0.0227130949, 0.0429330915, -0.17101869, 0.116467908, 0.116578884, 0.0260287896, -0.0962790847, 0.036279276, -0.0381992906, 0.212093785, 0.158137083, -0.112858787, -0.131867021, -0.191359714, -0.146997213, -0.000313639641, -0.003441751, -0.0417472273, -0.0491207764, -0.178802773, -0.0664816052, -0.0104046613, -0.0142799169, -0.188737929, -0.0185466558, -0.0352328829, 0.0682502836, 0.0788259357, -0.195347801, 0.203497171, -0.154879391, -0.18561314, -0.17881757, -0.117247216, 0.0698423609, 0.0224083364, -0.0493452102, -0.140239567, -0.183991462, -0.113582537, 0.0816551074, -0.203832656, 0.148944646, 0.166977555, -0.168197036, -0.0038562566, 0.0320169367, -0.17292963, -0.15642412, -0.165192544, 0.182672083, -0.15258047, 0.101091012, 0.174555406, 0.0823695511, 0.157132462, -0.129125595, 0.0654330179, -0.166881204, 0.0782062784, -0.0887168273, 0.00821068604, 0.0453969091, 0.220597595, -0.196104899, -0.0166419595, -0.0927555114, -0.107461981, 0.221482277, 0.223973781, -0.0611179322, -0.0668021888, -0.0858261585, 0.0375918262, 0.267744839, -0.0345278829, 0.254966795, -0.00994786248, 0.022099562, -0.127365038, 0.18192032, 0.0513121448, -0.110994041, 0.25041303, 0.196979046, 0.135527775, -0.0681474656, -0.0267207474, -0.199583828, -0.0502842888, 0.00327560958, -0.0646822006, 0.19758679, 0.261831164, 0.0999355987, 0.0594527014, -0.154063612, 0.0252208039, 0.221329957, 0.131121457, 0.00249284413, -0.0733978972, 0.100284182, 0.0556562096, -0.0429260246, 0.0306841414, 0.219935, 0.13371262, -0.00598191097, -0.132255256, 0.221873939, -0.163495034, -0.0360863805, 0.0824131444, -0.239943579, 0.172781795, -0.212151602, 0.236218229, -0.0616496243, -0.0723682791, -0.0943582132, -0.173591569, -0.158820465, -0.0388342962, 0.209313601, 0.105139598, -0.0127423787, 0.23334001, 0.105608903, 0.189134374, 0.161174685, -0.0848595649, -0.13802968, -0.00375816296, 0.102438428, 0.0600083843, -0.197466984, -0.15549612, -0.0712063238, 0.154483199, -0.0873283222, 0.15228495, -0.0364889465, 0.179233074, 0.14827925, 0.185523212, 0.27177012, -0.0103518441, 0.156902194, -0.0411169007, 0.0607469641, -0.0220632553, -0.0432856232, 0.142093897, -0.147602007, 0.18813391, 0.0621521808, -0.181282967, 0.0722836629, 0.179992348, 0.0792825669, 0.247705981, 0.228616223, -0.0473009236, 0.00126909569, 0.0863893405, 0.155630812, -0.100628406, -0.123317964, -0.11671751, 0.0799793229, -0.16633673, 0.0691096857, -0.0983060077, 0.161242321, 0.171100721, 0.143575251, 0.182359606, 0.00890773162, 0.110979609, 0.0892734379, -0.105653889, 0.227419034, -0.03998366, -0.124580286, 0.130855098, -0.0131535288, 0.272792101, 0.179608643, -0.210909322, 0.00432928372, 0.21848838, 0.253688663, 0.106119879, 0.0625382364, -0.143925086, -0.0632008985, 0.0975730494, -0.141114861, 0.0668569505, -0.0672182292, 0.162051871, -0.122773834, -0.0107828472, 0.0403296016, -0.0795900598, 0.277176142, 0.00853289384, 0.173946515, 0.117141366, 0.183931693, -0.0793479383, -0.0215559229, 0.187337711, 0.061015863, 0.0663154572, 0.169271708, -0.201445878, -0.0256252605, 0.244238496, -0.231323823, 0.0469608344, -0.0628846064, -0.14439863, 0.113650277, 0.163789138, 0.021281559, -0.103731513, -0.192868605, 0.147293687, 0.0449895933, -0.160115749, 0.0899030939, -0.165846884, 0.198117554, -0.167129472, 0.218909174, -0.171495542, -0.161191314, 0.129484773, 0.0846461579, 0.169623926, 0.0230460148, -0.112478353, -0.0921991095, 0.211257413, -0.0030605495, 0.0351988226, -0.0332586169, 0.139157876, 0.0921685547, 0.122303888, 0.0700193793, 0.179862246, 0.0254115313, 0.204242676, 0.0813357979, -0.0274808407, 0.200144112, -0.119426139, 0.161797479, 0.0829108208, -0.153130651, -0.0846347809, 0.0271065533, 0.140034661, -0.130517483, -0.186353624, -0.0104580438, -0.201147348, 0.075118795, -0.045870319, 0.156480566, 0.0903002545, -0.00378783746, 0.192498252, -0.038612958, -0.131505221, -0.0437254906, -0.101072744, -0.0389576852, -0.164237425, -0.175792545, 0.0373107754, -0.119521856, -0.156602532, -0.113795958, 0.112055942, 0.113850042, 0.00677617686, -0.0850653872, -0.0733917803, 0.187380284, 0.182089031, -0.0248251855, 0.163996622, 0.132685319, 0.142668948, 0.0152747529, -0.0172108244, 0.216359109, 0.118470624, 0.123126626, -0.100131035, -0.054644499, -0.133699596, -0.0788406134, 0.115421988, 0.143789545, 0.187183872, 0.167815328, 0.202092215, -0.0217228085, 0.144933701, 0.106362499, 0.259433448, 0.15671441, -0.0946840271, -0.186438739, 0.0081841452, -0.14182502, -0.00946078729, -0.0603948757, -0.00157379068, -0.18708539, -0.0983730108, 0.0651348308, 0.00732422806, -0.0354584157, 0.0694651306, -0.170068949, -0.146637738, -0.0188922025, 0.130627021, 0.253977299, 0.161411852, 0.247188866, 0.203512952, 0.0883074552, 0.113822445, -0.046621304, 0.175482243, -0.0289865751, -0.15941821, 0.178795829, -0.277471334, -0.199458614, -0.00665188488, -0.127981231, -0.209003299, -0.148039356, 0.137913957, 0.0634118468, 0.166315272, 0.170956552, -0.215199739, -0.110592142, 0.0109336888, -0.026153028, 0.0884291679, -0.0187547766, -0.0606251135, 0.185180321, 0.139575243, 0.104148917, -0.216128081, -0.0651518703, 0.100283109, -0.0865191743, -0.0341802686, 0.0216208063, 0.072604768, -0.122850962, -0.0247077513, -0.147178918, 0.12824367, 0.182407543, -0.000500810798, -0.184659287, -0.0473984033, 0.0934755877, -0.0367431417, -0.15300943, 0.24329026, -0.151669785, -0.114891134, -0.186268806, -0.0633910894, -0.166982651, -0.107574888, -0.0891585425, -0.139917731, -0.0927230418, -0.175722167, -0.0773153529, -0.115566179, -0.145081356, -0.147527725, -0.138250202, 0.217643395, 0.224325195, 0.150407761, 0.0212292019, 0.0613440573, -0.188086301, 0.23438555, -0.0300599616, 0.206930742, 0.0815451145, -0.375011235, -0.0562498868, 0.00639961939, -0.0058033783, 0.168399513, -0.0654805675, -0.0274477936, -0.109949432, -0.0414189361, -0.0130247008, -0.200141788, -0.163074657, -0.170476168, 0.193809062, -0.111856036, 0.152590171, 0.0143048586, 0.185440674, -0.169017375, -0.158529475, 0.00929309428, -0.0942657292, -0.148064896, -0.134354785, -0.206875667, 0.202413216, -0.0598236918, -0.166547075, 0.152515814, -0.163616508, -0.202204078, 0.114426211, -0.182107091, 0.0707437545, -0.0522488952, 0.0869736522, 0.0402545184, -0.0945940241, 0.185991451, -0.124674715, -0.03174752, 0.162187114, -0.137566179, 0.184869885, 0.0221520253, -0.197971106, -0.170951381, 0.0330120921, 0.0279635787, -0.139334649, 0.0697774142, -0.197592616, 0.17985791, -0.0284902453, 0.115595266, -0.201338783, 0.0367098935, 0.07913436, 0.127372906, -0.124858603, -0.0313890874, -0.181075796, 0.0527459234, -0.135128409, 0.0876705199, -0.184465155, -0.0735049844, 0.0535863489, 0.00994851347, 0.137904853, 0.0959903747, -0.186176807, -0.0812415555, -0.112533055, 0.174689725, -0.096371375, 0.122750133, -0.0395515561, -0.0953361019, -0.142940253, 0.0410725772, 0.111044452, 0.0270516891, 0.161732242, 0.0858138651, 0.0895572454, 0.037848372, 0.162806571, -0.0460997261, 0.0349680036, 0.160732448, -0.129507929, 0.113114722, -0.0166504215, 0.120835945, -0.0622817799, -0.133667618, -0.0202337652, -0.0207774434, 0.170200497, 0.00774796167, -0.0592490025, 0.230593592, -0.00738770561, -0.0436120033, -0.0423453487, -0.0329519622, 0.206478819, 0.0155085847, -0.0256422833, 0.0234079231, 0.0186074525, -0.1795073, -0.180009589, -0.00913083926, 0.196808264, -0.21870546, -0.179154739, -0.0917448699, 0.14978005, -0.061042279, 0.012972462, -0.0826573893, -0.0671150908, -0.138860673, 0.00231725769, -0.166636378, -0.0871414915, -0.0446091257, 0.192121252, -0.109329425, 0.0788124055, 0.152980164, -0.129419059, -0.0276356209, -0.0259925574, -0.0593720526, 0.179485679, 0.0266083553, 0.0747748911, 0.101830587, -0.0766663998, 0.0163841695, -0.161232248, 0.0171750262, -0.279156268, 0.221496373, -0.186395198, -0.0143639594, -0.143523067, -0.0878556073, -0.0815294832, -0.067358315, -0.16824618, 0.111157678, -0.160450444, -0.161506832, -0.0405490361, 0.102888331, 0.0339654423, 0.118124977, -0.00176335871, 0.165163413, -0.0700196028, -0.00438803434, 0.175777838, 0.186697081, -0.121123411, 0.122397795, -0.0532331169, 0.0590221882, -0.105305605, -0.204723135, -0.175872728, -0.0677143931, -0.161616057, 0.0188506059, -0.210944623, -0.148904279, -0.113570303, 0.221049219, 0.0313297138, 0.107811853, -0.180402234, 0.109366827, 0.0825608298, -0.15245305, 0.205485806, 0.0317764021, 0.0504349619, 0.00149199367, 0.00595451333, -0.174039871, -0.0160308499, 0.194607705, 0.179732472, 0.0789086595, 0.197504297, 0.0629399493, -0.116470531, -0.186572343, -0.0899397954, 0.19567205, -0.00335924979, -0.208514586, 0.0973969102, 0.0326924175, -0.206587866, -0.0218385514, 0.0725486577, 0.155927837, -0.188840836, 0.0960423201, -0.165740326, 0.1604902, 0.267009914, 0.0818572193, 0.260096461, -0.186999142, -0.0683261901, 0.0665122792, 0.0479869246, -0.101161063, -0.0638602898, -0.218564659, -0.0387957096, 0.0902684554, -0.16147168, -0.0608646087, 0.062403813, 0.0504773445, 0.0787408352, -0.0066665113, -0.0551999062, -0.200761631, 0.00933836773, 0.297097772, 0.16794759, -0.185238838, -0.0823579729, 0.0469955355, 0.3021909, -0.134364396, 0.196597978, 0.0334144868, 0.0336058177, -0.10905616, 0.0721478015, 0.0315832756, 0.189071074, 0.0691891909, 0.34283489, 0.150725141, 0.00169667602, -0.117639907, 0.121499099, 0.194060832, 0.0223687626, 0.161883071, 0.516069353, 0.384240836, -0.0662594065, -0.219141394, 0.113189861, 0.174268171, -0.0602926537, 0.023207292, -0.0562035777, 0.223606259, 0.17101483, 0.15739201, -0.0148757435, 0.195277646, 0.0899973437, 0.48358345, -0.0253587756, -0.00797794759, -0.0891540423, 0.092290625, -0.185479164, 0.0852196366, 0.213107035, 0.0252361298, 0.200780615, -0.189653561, -0.182161033, 0.021594137, 0.145947233, -0.112602293, 0.0719485134, 0.073290661, -0.068946287, 0.146695599, -0.164526656, -0.0765778124, -0.171564609, -0.0508742183, 0.214564845, -0.203749716, -0.138006911, -0.0141354799, -0.206376866, -0.174090385, -0.0728472918, -0.0598603934, 0.0906234831, -0.216011941, 0.122935966, 0.127648816, -0.192449927, 0.0749056488, 0.138052747, 0.105709121, 0.0347812921, 0.110028967, -0.135962948, -0.144907042, 0.154864535, 0.0592765659, 0.0534629077, 0.0385289937, -0.156602025, -0.0317876786, 0.208689615, 0.177388117, 0.00780889392, 0.0349562615, -0.0682702363, -0.0363424569, -0.0553218275, 0.133666351, 0.00441069901, 0.096022442, -0.133351326, -0.00378321111, -0.136954084, 0.0019338131, -0.181480229, -0.155208886, 0.203421369, -0.125472635, -0.171183765, -0.165254846, -0.133507237, -0.0173198301, 0.21947293, 0.143755376, -0.0401268005, 0.0731849745, 0.0850220844, 0.0371454805, -0.0326308534, -0.0790177658, 0.0200932287, -0.121129356, -0.126217842, 0.0199649576, -0.169905156, 0.237343252, 0.177157223, 0.165131941, -0.183802426, -0.125728503, -0.134026647, 0.102495909, 0.0696081296, -0.167917982, -0.166213095, 0.0101573337, 0.134656668, 0.0390270464, 0.147898167, -0.0125229191, -0.171897367, 0.18344982, -0.0810840577, -0.00678340718, 0.122303508, 0.0799789727, -0.0815866068, 0.0310235824, 0.154979914, 0.0764822215, -0.128525659, 0.152218923, 0.0648555607, 0.10429927, 0.165912151, -0.00706859026, -0.0883911997, 0.165610254, -0.205627054, 0.172161713, 0.206336021, 0.121359043, 0.0919625983, 0.223842055, -0.209351197, 0.0634121448, 0.227562383, 0.0355994329, 0.00256789825, 0.237201974, 0.037827909, -0.177561209, 0.222521156, -0.202093512, -0.0229218453, -0.118946023, 0.0302829295, -0.0116465688, 0.022469908, -0.211659819, 0.0230853111, 0.193522528, -0.0245168656, -0.201854825, -0.0753775686, -0.0310619175, -0.200594962, -0.0756556392, -0.128971279, 0.156894669, -0.179421097, 0.0251898766, 0.023289308, 0.0580800325, 0.140855506, -0.0611620098, -0.0153288692, -0.00615723431, -0.21604234, -0.084130466, -0.15956971, -0.0087262094, 0.0838872939, -0.0140172839, -0.186466902, -0.0742408633, 0.134943053, 0.0629239827, -0.158630103, -0.111521803, 0.00854839385, -0.152197734, -0.187499329, -0.146150753, -0.0487617552, -0.12666437, 0.148413315, 0.00076122582, -0.0748235434, 0.210751161, 0.0419287831, 0.0125453025, -0.0107841194, -0.07289505, -0.126931146, 0.140740082, 0.129911378, -0.0123122483, -0.202497944, 0.214250848, -0.119241752, -0.205320999, -0.152010053, 0.159491345, -0.165408313, -0.185733244, 0.0348138064, 0.191792235, 0.200777933, 0.161115959, 0.115620837, -0.125909343, -0.0419274867, -0.0674549639, -0.164896861, 0.200165018, -0.163343281, 0.133848891, 0.066679135, 0.0242425203, -0.215839475, -0.177766964, -0.178671584, 0.179792449, 0.210112378, 0.118905827, 0.180896834, -0.202173829, 0.175342038, -0.0985738114, 0.193638191, 0.0229219347, -0.0222909003, -0.0943710357, -0.024797678, -0.16884923, 0.0664104372, -0.0999937505, 0.0858398229, 0.203513905, 0.182638362, -0.0276584178, 0.143701836, -0.159802675, 0.138917372, -0.0687357336, -0.118034951, 0.165999964, -0.0323487371, 0.123346254, 0.0527410358, 0.137795433, 0.01838772, 0.0875368267, 0.173462018, -0.0463278592, 0.129204765, 0.150611833, 0.107375845, -0.0264342129, 0.169134393, -0.0467272401, 0.199903682, -0.0980908126, -0.190550029, -0.0762602538, -0.0315628797, -0.0798259974, 0.160073265, -0.00462961197, -0.183606789, -0.0188505352, 0.0691810995, -0.197972029, -0.15645048, 0.116300687, -0.124517485, 0.173053637, 0.0755809918, 0.081306681, 0.161437288, -0.0970465466, -0.130220771, -0.0481538028, 0.180401117, -0.0649009943, -0.165097132, -0.130503684, -0.00572030758, 0.0470085293, 0.00363709033, 0.00171510922, 0.0857786089, -0.0651379302, -0.066770114, -0.157249182, -0.17459558, 0.108071186, 0.18482846, -0.0944221914, 0.0439717509, 0.0515320636, -0.101472825, -0.191481218, -0.157240301, -0.0539558493, -0.125500441, -0.157671779, 0.217446938, -0.153299645, -0.0213545188, 0.169633135, -0.202749312, 0.15830192, 0.123832054, 0.202120841, 0.178851813, 0.0410678647, 0.00611580582, -0.053331662, 0.0464291424, -0.0324332118, -0.106219634, -0.216207579, 0.228908926, -0.0941737071, -0.134803563, -0.202760994, -0.00565075129, 0.168043837, 0.0981038436, 0.0794638395, 0.167057589, 0.128910467, -0.0112976059, 0.170332775, 0.0585579872, -0.22341539, 0.0355694294, -0.154355466, 0.0759388655, 0.105432287, -0.0729613379, -0.0318719745, -0.0295223258, -0.100262426, -0.100136787, -0.0460873507, -0.0712981075, -0.0222990401, 0.0588900596, -0.113420017, 0.17419365, -0.10283038, -0.144499213, 0.124155849, 0.0594922118, 0.0716532618, 0.129410103, 0.0517303199, 0.148354009, 0.0255827624, 0.0190704111, -0.149046123, 0.136326805, 0.105247073, -0.0295574721, -0.238865554, 0.0468696915, 0.0912098587, 0.0714069828, 0.0229250956, 0.110962324, 0.131823346, -0.165668309, -0.00778792799, -0.185458347, 0.20212841, -0.0874781683, 0.0586535111, 0.143871352, 0.275070757, -0.044842042, -0.0718936771, -0.072808072, 0.0834283978, 0.133895293, 0.198372915, -0.0804026723, 0.188191667, 0.0981120318, 0.206251636, 0.177413091, -0.102985151, 0.196867242, -0.013884523, -0.188111216, -0.130392522, 0.0190863628, -0.148793653, -0.0467367023, -0.192909583, -0.0972905159, -0.137692288, 0.211145386, 0.140261218, -0.142052516, -0.194741502, 0.192499146, -0.049346976, 0.0810934156, 0.0646863505, 0.125058278, -0.0799507052, 0.132487938, -0.0906506926, -0.0655713826, 0.0928521007, 0.183620468, 0.138887301, 0.162195206, 0.155351385, -0.058083415, -0.0219758153, 0.0991288573, 0.0169533193, 0.103431225, -0.130349159, 0.0779341757, -0.241531909, -0.178271845, -0.138706401, -0.0624510534, 0.111244112, 0.111007653, -0.0359138511, 0.0459302366, 0.0223376025, 0.165935397, 0.0252500176, -0.147416338, -0.110299625, 0.00361161027, 0.167947292, 0.132642567, -0.0257409364, 0.250626832, 0.08315216, 0.0183384717, 0.0648797005, 0.108391851, -0.218746424, 0.223503336, 0.0558422469, 0.081787914, -0.0234055668, 0.0559378527, 0.0436194129, 0.0106922649, -0.0692483187, -0.0691979155, -0.0494184643, 0.0244371723, -0.167693228, 0.158963591, -0.115475364, -0.173542932, 0.0758400708, 0.0158745944, 0.176581964, -0.032615751, 0.140387014, -0.0867669731, -0.0148333311, 0.0844656676, 0.191718534, -0.194510147, -0.0462476611, -0.142200023, -0.127892822, -0.0507825464, 0.0212071091, 0.0735275894, 0.101716116, 0.074662827, -0.197910756, -0.133237764, -0.187822059, 0.145099476, 0.0327065587, -0.146056384, -0.0505298674, 0.108181708, 0.107639544, -0.138911337, 0.122266933, 0.115411207, 0.144105688, 0.0382299572, -0.148832917, 0.139190271, 0.167309538, -0.144928098, -0.0563678443, -0.043597877, -0.1119316, -0.12973395, 0.0584410578, -0.0437880307, -0.0104946736, -0.165186569, -0.0112327933, 0.118900821, 0.182406887, 0.192648664, -0.00062443316, -0.184834018, 0.199227616, -0.121603794, -0.167943582, -0.00912922435, -0.0713112056, 0.171490803, -0.0891723186, -0.0559416711, 0.174898937, -0.070852831, 0.0793064982, -0.212293357, 0.0701971725, -0.0021967846, 0.0451571047, 0.0195722282, 0.0461180322, -0.00641624769, 0.0517838448, 0.137161285, -0.0997539088, -0.118641637, 0.234035909, 0.150188163, 0.0618825108, 0.0109362891, 0.0320615731, -0.1136159, 0.0582003295, -0.195525587, 0.137793392, -0.0844204947, 0.0396005958, 0.207778886, 0.199851304, -0.0735878795, 0.106541574, -0.0736700818, 0.13129513, -0.0877129585, -0.0679071546, -0.0147504732, 0.202523276, 0.194757164, 0.0617246218, -0.123547576, -0.248862714, 0.104788274, -0.100657925, 0.000960324774, 0.188817993, -0.108579315, -0.204805076, -0.244371086, -0.0309919175, -0.00391102675, 0.070959501, -0.016308561, 0.146207169, -0.172038585, -0.13708587, 0.14507246, -0.0678439513, -0.154684559, -0.240108371, 0.138188958, -0.206409857, -0.159489393, -0.214073613, 0.107187405, -0.204427004, 0.0283892639, 0.172533706, -0.206037849, -0.11586225, -0.24410139, 0.109407388, -0.0316474549, 0.158885717, -0.0667252243, 0.118405201, 0.289276123, -0.165092245, 0.108930469, 0.070623219, 0.179036945, 0.108090542, 0.182895318, -0.156233117, -0.117184833, 0.142791912, -0.0148069672, -0.0239627529, -0.214217961, 0.137310907, -0.188492745, -0.246256724, 0.147092804, 0.176855475, -0.0857564658, 0.0680939779, -0.0448941737, 0.0981446952, -0.172164232, 0.304895014, 0.0906158388, 0.297383636, 0.0652368665, -0.0184425749, 0.28164503, -0.173171684, -0.238063306, 0.186662257, -0.00241088937, 0.125462785, 0.304029018, -0.342890888, -0.0287288111, 0.17390269, -0.066968292, -0.177149415, -0.0643516853, 0.122750431, -0.0577152073, 0.0959472433, -0.0236832555, 0.116106987, -0.160913095, -0.0329174101, -0.014049178, 0.123443589, -0.0367398858, -0.110727645, 0.15123257, -0.144489914, 0.0620885342, -0.191643208, -0.0555331744, -0.0333120152, 0.0111381225, 0.200533777, 0.188959613, -0.155872673, 0.0341290683, -0.192276001, -0.171046734, -0.0678890795, 0.0327494256, -0.123621963, -0.123488769, 0.00637859805, -0.0630104989, 0.205584362, 0.169972613, 0.0232409332, -0.0955383033, -0.102426589, -0.0347150117, -0.141734734, 0.128293246, -0.0925778523, -0.0108686425, -0.13012214, 0.0815413147, -0.0893505439, 0.0880092233, 0.02950003, 0.23860997, 0.183169857, -0.0187763385, -0.13275674, 0.234897241, 0.110683218, -0.18547368, 0.144646749, -0.074404262, -0.10398934, -0.135641322, -0.157735169, -0.124934033, 0.137574792, -0.0147348205, -0.139187038, -0.221444562, 0.107474491, -0.156930476, 0.0779651478, 0.0951431543, 0.0451893285, 0.0516319498, -0.191372216, 0.0186820943, 0.126253679, 0.042005375, -0.0644702911, 0.114736617, 0.16525045, 0.116882309, 0.070220463, 0.188503683, 0.102188125, -0.0785993859, -0.15001981, -0.0465400182, 0.231806532, 0.0954680666, -0.184053317, -0.0501416922, 0.167674035, 0.191605791, -0.0193787068, 0.0830391496, -0.107822374, 0.207061484, 0.0861738399, -0.00507401815, -0.00288677309, 0.00758164329, 0.121445261, 0.092905201, -0.163787112, -0.0633125082, -0.123845324, 0.0347361527, 0.0725645497, 0.254036367, -0.0882892832, 0.199529752, -0.203118846, 0.0343604796, 0.198467344, -0.235339314, 0.237031609, 0.0543105453, 0.153027922, -0.00393469399, 0.10333398, -0.0708734468, 0.0561602749, -0.239301354, 0.0680253059, 0.183111206, 0.0810918957, 0.24312824, -0.160712034, -0.137365401, 0.21149838, -0.208581164, 0.0860498995, -0.222985104, 0.195945591, 0.0468437523, 0.0805253461, 0.301470578, 0.110695809, -0.153531685, -0.107340924, -0.115410239, 0.0342867225, 0.195745423, 0.0319843628, -0.207723111, -0.0392347164, 0.231147945, -0.129315481, -0.176766947, 0.177469, 0.192669258, -0.226546422, 0.0189814288, 0.0556515306, 0.107801184, -0.265750676, 0.168204769, -0.0855395198, -0.059515968, 0.0842674077, -0.0828177929, -0.130357698, -0.184084356, 0.137147471, 0.0251989067, 0.190306425, -0.209870204, -0.0716328025, 0.0316385627, 0.153478116, 0.396686941, 0.147947639, 0.192033961, -0.0293983817, -0.206629544, 0.275531769, 0.46042946, 0.140281811, 0.24135609, 0.0912894011, -0.17723383, -0.0607077032, 0.0781214163, 0.374888659, 0.137123927, 0.672217488, 0.276213497, 0.175734013, 0.0280658901, 0.0311749578, 0.0746272653, 0.349832982, 0.218783423, -0.185958922, 0.68218708, 0.800624728, 0.210476741, -0.00437949831, 0.130500868, 0.0502584949, 0.0294641983, -0.0176065117, 0.108612187, 0.358226597, -0.121234097, 0.108403966, 0.231736287, 0.210347712, -0.0159039721, 0.554084659, -0.167776093, -0.0969910622, 0.255162835, -0.0156714115, 0.26939097, 0.0617705248, -0.0752833113, -0.0614468567, 0.0244390815, -0.091742225, -0.137374878, 0.0531701297, -0.174850404, 0.141812295, -0.150860801, -0.187058046, -0.0874524713, -0.0264754221, 0.140813321, 0.182697207, -0.153970152, -0.177734926, -0.141945884, 0.0117159495, -0.00985656679, -0.00101221201, -0.0196746346, -0.174091488, -0.052107349, -0.22018443, 0.14820832, 0.0818826631, 0.233457372, 0.0977712348, -0.115955748, -0.0530783907, -0.140831947, 0.122053191, 0.121684685, 0.264127553, 0.0270333346, -0.0565839447, 0.019359095, -0.194519073, -0.00262582256, 0.0962572768, 0.0432850756, 0.113889135, -0.0236177016, 0.236521289, 0.183020383, 0.123297013, -0.167065337, 0.191284567, 0.14299646, 0.0509699844, -0.0904205814, 0.110933594, -0.0448181033, -0.187609032, -0.0712240487, 0.176699147, -0.118739776, 0.271520019, -0.166733369, -0.165289536, -0.0146756694, -0.00527196797, -0.0271551386, 0.00151156972, 0.228332981, -0.0739963129, -0.15750289, -0.0617005788, 0.00474839332, -0.154549867, -0.106653541, 0.176194146, -0.126685426, -0.0473142527, -0.0840078592, -0.00723607512, -0.212898895, 0.168081641, -0.185128301, -0.0536887795, 0.0943454057, 0.182923332, -0.0643337741, 0.196476832, -0.151796073, -0.0726564005, -0.0456830412, -0.0407369286, 0.192159489, -0.025926657, 0.0753762797, 0.0520100966, -0.0740965158, -0.0278436802, -0.0877467319, -0.213060349, 0.0216137562, 0.013314412, 0.175274462, 0.137478024, 0.0799314231, -0.00686348975, -0.124030545, -0.0374336392, 0.0357716046, -0.103798419, -0.0145825977, 0.123516023, 0.147583932, -0.0383550748, 0.0558126122, 0.107982129, 0.20239383, -0.106662877, -0.186953425, -0.145417884, -0.153639495, 0.027993679, 0.190795079, 0.0476124473, -0.12085294, -0.109654099, 0.167916715, 0.200663969, -0.00801608246, 0.0825436339, -0.0943990722, 0.113534227, 0.17334342, 0.111058161, -0.124200851, -0.0368134826, -0.00652719568, -0.141232178, -0.0518599898, -0.0585245639, 0.0653005391, -0.235346124, -0.148109958, -0.133401841, -0.114027344, -0.0275279973, 0.0593129881, 0.0982646197, 0.0619096607, 0.0287333895, -0.0120723862, 0.217594147, -0.139917493, 0.167802855, -0.168642655, 0.0747052282, 0.269419819, -0.116047248, -0.00862775743, -0.221282467, -0.118697263, -0.205058426, 0.093385309, -0.101342008, -0.183804184, -0.0605899505, 0.121015184, 0.0115664136, -0.208521381, 0.170277372, -0.0868665427, 0.248344138, -0.0432597287, 0.0541927218, 0.174610093, 0.181111693, 0.0449905209, 0.108599983, -0.130895346, 0.00717880577, -0.129434913, -0.042265553, 0.144251227, 0.259774655, 0.186873987, -0.0417911112, -0.048804868, -0.0295425355, 0.191073224, 0.0611833222, -0.0762384161, 0.140305713, 0.123962991, -0.0918691456, 0.218360201, -0.117257692, -0.127649173, -0.0255799256, 0.0222741216, 0.104327299, -0.0732962042, 0.0868302435, 0.228259474, 0.213780165, -0.0154352821, 0.131837606, 0.23168534, -0.214955419, -0.172440171, -0.0347957499, 0.128808409, -0.126937971, 0.061891485, -0.0297385268, -0.111321308, -0.0260849223, 0.120274864, 0.109222718, 0.0718200356, -0.235081047, 0.149947703, 0.0434079766, 0.0383607633, 0.116888225, 0.140750632, -0.0997844785, 0.174422219, -0.138142154, -0.0749339536, 0.0785625502, 0.120397143, -0.160959065, 0.0388336182, -0.167576253, 0.28271389, -0.191148162, -0.0925715864, 0.183668092, 0.0161793791, -0.0543912798, -0.0963794515, -0.102523632, 0.0610520095, 0.219306812, 0.0398645885, -0.0823789462, -0.102402054, 0.0275531858, 0.0220897496, 0.00813651085, 0.224854186, 0.173899412, -0.0672621354, -0.160013005, 0.224919304, 0.156423524, 0.0298209954, 0.127081707, 0.0212131441, 0.0445396155, 0.0335416645, 0.108812883, 0.111677632, 0.198874697, 0.0437096506, -0.165222168, 0.146299198, -0.0258866847, 0.206391677, 0.21082823, -0.125449836, 0.212311164, 0.166904435, -0.0247623175, -0.0211795866, 0.0768647045, 0.200587884, -0.0911418498, -0.169951767, -0.160309315, -0.0806967169, -0.158640265, 0.113370135, -0.00294652581, 0.0389382094, -0.216152698, -0.0083335489, 0.0735277981, 0.0742935687, 0.128101602, -0.00542548299, -0.115529254, 0.113532469, -0.160332292, 0.0508067459, 0.0624400526, 0.209660366, -0.214744583, -0.092242986, -0.160066396, 0.153950915, -0.212624639, -0.136968851, -0.135505289, 0.121049806, 0.0121994615, 0.151701763, -0.11071489, -0.171668932, -0.0537894666, -0.0878971219, -0.205776945, 0.099695608, -0.190786853, 0.0116519928, -0.144893363, 0.0865933746, 0.123252288, -0.182795584, -0.187821805, -0.18338947, -0.205582917, -0.0606609881, 0.0743346661, -0.0960690454, -0.211429507, -0.0481314957, 0.135181442, -0.216266423, -0.0187025368, 0.0537178665, -0.108392335, 0.0977317542, 0.129478082, 0.0895232707, 0.0533473045, -0.0970297307, -0.206168756, -0.139258206, -0.0563539565, -0.131601334, -0.0870515406, -0.0619503707, 0.20224908, 0.189971015, 0.208698735, -0.0417911559, -0.0538787693, -0.0976427495, -0.00286698341, -0.0744511336, 0.0304896683, 0.0333309472, 0.0902835578, -0.0216697603, 0.0137269134, 0.150900915, -0.182306468, -0.20932512, 0.0233798623, 0.136948779, 0.0849334449, -0.092384629, 0.188453048, -0.0954338461, 0.0955692083, -0.00602588151, -0.182517394, 0.0109124696, 0.106711015, -0.203821674, -0.108474381, 0.118665077, 0.153626904, 0.0262012091, 0.0375920273, 0.154369608, 0.0770949274, -0.117124625, -0.0335433446, 0.0450399965, -0.128809497, -0.00421985984, -0.0802144259, -0.139152095, -0.153811246, -0.120795593, 0.143708199, 0.185526088, -0.142273381, -0.195421949, 0.152865365, 0.0122631425, -0.000951811671, 0.0673113987, 0.136099085, -0.0278965831, -0.0474108718, 0.213819981, 0.142901793, 0.00495843589, 0.0418358333, -0.00355575676, -0.0105182827, 0.16393365, 0.101665772, -0.169067964, -0.195942327, -0.0434645265, 0.0727494806, -0.198469073, 0.132359818, 0.0526619218, 0.0468863398, 0.134476244, 0.0864710659, -0.16446723, 0.0303983875, 0.0437866561, 0.16037491, 0.161007166, 0.0387010314, -0.202730685, 0.044473853, -0.129946947, -0.05610618, 0.164238542, 0.137609839, -0.208719894, 0.153201148, 0.13046816, 0.180548891, 0.156915024, 0.205377564, 0.0167820454, -0.11153812, -0.0215259828, -0.126827091, 0.162156314, -0.0532439612, 0.0574748926, 0.0771525949, -0.0153041324, -0.0292977095, 0.191961616, -0.0606812425, 0.0860238746, -0.146850556, -0.0733355656, -0.149648055, -0.0798214898, 0.0446455069, -0.170179084, 0.0201480612, -0.0888226479, -0.103910781, 0.119667917, 0.153799519, 0.054285761, -0.148660555, 0.035269402, 0.109882556, 0.204186887, 0.0496170707, 0.161113545, -0.135843858, 0.253733486, -0.0944817513, 0.0327358693, 0.230729103, 0.108584575, -0.221280649, -0.11051406, -0.145698979, -0.132175505, 0.178192541, -0.156799883, -0.137536705, -0.0399425589, -0.134871528, 0.18148458, 0.11162968, 0.092132248, -0.171199903, -0.0500270128, -0.191958666, 0.122761637, 0.114319079, -0.13137719, -0.0537062585, 0.113184899, -0.263052046, 0.141020328, 0.239564508, 0.170219958, 0.102902547, -0.101794772, 0.158655852, 0.161232308, 0.257718861, 0.234837502, 0.0273188651, 0.121293917, 0.120111875, 0.256624699, -0.0763987452, 0.0835199878, -0.0190323666, -0.103317492, 0.0232522283, 0.10880886, -0.0914563537, 0.109213397, -0.0964482874, -0.169531703, 0.281256527, 0.0533225201, -0.00718479324, -0.117911838, 0.0900024846, 0.135364503, -0.0926576406, -0.165947258, 0.212630153, -0.199972525, 0.206199676, 0.18481414, -0.179684758, 0.0156940166, 0.11673253, 0.173709407, 0.145675406, -0.00235269964, 0.186596662, 0.211974829, 0.000806359749, 0.0446996912, 0.0769063011, 0.0293873399, -0.0577886961, -0.0997519717, 0.115017757, 0.0576308221, 0.0125924861, 0.225485265, -0.00981596857, 0.139237881, -0.0530043356, 0.260116875, -0.22942251, 0.0249016378, -0.0571197607, 0.153768301, -0.206047684, 0.0895582587, -0.279679924, -0.0219289549, 0.10167665, 0.0845968127, 0.00727231754, -0.0432331599, 0.225695342, -0.0686216056, 0.28638041, 0.272146463, 0.140005305, -0.0245791562, 0.0761088356, 0.201061755, 0.00954514742, 0.218374774, -0.168220788, 0.103706576, -0.20218125, 0.0332696922, -0.0424223542, 0.108355887, 0.1041262, -0.00260003889, 0.0343024097, -0.102693766, -0.100874119, -0.0986998156, -0.235685483, -0.0899084508, 0.0854150206, 0.0691602379, -0.185052946, 0.0787002891, -0.165196121, -0.0326854065, 0.0315757096, -0.149115399, 0.0719742849, 0.0407750756, -0.0767336041, -0.187577948, -0.048541002, 0.0360414013, 0.249366537, -0.192914456, 0.190689608, 0.0374177843, -0.0437144637, 0.213710159, 0.096700497, 0.00223939074, -0.0764921829, -0.0575337037, -0.145044506, -0.0802579448, 0.064725399, 0.0837969631, 0.0941284671, 0.0538992845, -0.0705573037, -0.115551233, 0.0803196281, 0.0834578872, 0.0238675773, 0.136617467, -0.186541721, -0.0417114496, 0.245139882, -0.00578208687, 0.0275053699, -0.0501771569, -0.179348543, 0.173432946, -0.0807827562, -0.179962143, 0.110388212, -0.146068901, 0.213116661, 0.144476965, 0.0446254946, 0.146554768, 0.093346484, 0.16855067, -0.192628831, -0.028239293, 0.160450786, 0.203553155, -0.11479301, -0.107505403, -0.0260372236, -0.144633308, 0.114200078, -0.127950758, -0.214850038, 0.207950816, -0.0725203902, 0.0758482069, -0.046793025, 0.0461012349, 0.0468173474, 0.00463971123, 0.0375378318, -0.0815252587, -0.0458168387, 0.10962835, 0.0194397829, 0.0926095471, 0.073319912, 0.0239949729, -0.0836053863, -0.137725636, 0.0898624137, 0.253191203, -0.192230299, 0.223583639, 0.214670718, 0.12229877, 0.229018718, -0.0431688577, 0.110472642, 0.139069289, -0.0282006748, 0.101184413, 0.0894554704, -0.0786872953, -0.0111689866, 0.0286502857, -0.0633932576, 0.171827883, -0.0444677696, -0.0850014165, -0.169253916, 0.120693155, 0.0252687819, -0.170735449, -0.123299576, 0.220411927, -0.217961624, -0.149791226, -0.171596184, 0.0943251699, -0.100113608, 0.087037079, 0.0855410993, 0.0791215971, 0.11918585, -0.0505308397, -0.117827907, 0.063941285, 0.00416628085, 0.0839637816, 0.267723888, -0.227810621, -0.0777227134, 0.0388324112, 0.256261855, 0.245122582, -0.138452694, 0.0876130164, 0.0878035948, 0.129902616, 0.102416001, 0.264991552, 0.139974669, -0.013653418, -0.065480873, 0.0472233519, -0.193420827, -0.0574077927, -0.100826748, 0.0330015197, 0.15693666, 0.109514177, 0.00890431553, 0.031340763, -0.0226426851, -0.170719773, 0.0925062895, -0.228847221, 0.130559415, -0.0788129494, 0.128267556, 0.176107913, -0.0924457237, 0.0958436653, 0.144238055, 0.0475376062, -0.100932501, -0.115049355, -0.207394749, 0.26449883, -0.0507705212, -0.0272947475, -0.00600530533, -0.106777452, -0.117991619, -0.234071791, 0.0523665883, -0.204911649, 0.043802131, 0.1575744, -0.220566079, 0.0123432605, 0.0531032309, 0.103713386, -0.205086485, 0.223250866, -0.0471659116, 0.00876451191, 0.214768395, 0.246275902, 0.0651466101, -0.197602212, 0.205826506, -0.0679371729, -0.000915050507, -0.105748199, -0.145877063, -0.201368526, 0.0879625231, -0.0965842009, 0.198548451, 0.161472961, 0.0642927736, -0.0918231159, 0.182744697, 0.0693864375, -0.188803703, 0.00650767982, 0.172555879, -0.0635101199, 0.00677795708, 0.202838168, 0.040710941, -0.209036991, -0.144217819, 0.188803896, -0.00212830305, -0.148173034, -0.20080778, -0.192079917, -0.0633593947, -0.16399309, 0.153926134, 0.203168228, 0.0955855399, -0.137954876, -0.19007811, 0.123448029, 0.21018137, -0.0810624957, -0.111288175, 0.021730572, 0.146542504, -0.157430366, 0.181623116, 0.126291782, 0.207365617, 0.165423319, -0.0239322782, -0.0631945282, 0.12825425, 0.200958624, -0.052633673, -0.0713848397, -0.185413659, -0.101239368, 0.182738468, 0.165163174, 0.0180790871, -0.15865013, -0.0937678143, 0.19551906, -0.0590572059, -0.0486637354, 0.0733446032, -0.0732812583, -0.0904489607, -0.0468690395, -0.124550417, -0.0455771685, -0.104021177, -0.185393631, 0.0408243984, 0.105959103, 0.119070217, -0.215867609, -0.12802428, 0.069313094, 0.0940398425, -0.179975063, -0.0170270354, -0.16964227, 0.0537156612, -0.0739964396, -0.210699499, -0.169508368, -0.114205375, 0.20856382, -0.0094743818, 0.023435086, 0.0358004421, 0.044800505, 0.186260834, 0.149650797, -0.101585321, -0.194993809, -0.0581209809, -0.189571068, 0.00125160813, 0.174607709, 0.0704791695, 0.140320167, -0.0318251103, -0.0955716968, 0.16221489, -0.177237138, -0.00738732517, -0.0435195267, -0.00547859073, -0.215163887, -0.00860790908, -0.00653317571, 0.126314595, -0.103846706, -0.0728396028, 0.0168418288, -0.0725217909, 0.109986708, 0.0920121819, -0.171025246, -0.0454324782, 0.0630950481, -0.0997218713, -0.0783640891, -0.00420938432, -0.18078503, 0.172304526, 0.125460967, -0.0567836761, 0.113854423, -0.00121866679, -0.0124422107, 0.037865255, 0.0818271786, -0.159302071, 0.0689702779, 0.16112043, 0.000206770215, 0.0466447026, -0.219438955, -5.96225691e-05, -0.000440880656, -0.174127713, 0.066909574, 0.0277200025, -0.213515118, 0.060687568, -0.0385784097, -0.109999962, 0.0165164806, -0.188594639, -0.0643988177, -0.0376132242, -0.113160878, -0.177742392, 0.20572792, 0.197053879, 0.178338304, 0.0188686363, -0.0623674206, 0.0213672761, 0.165976256, -0.0983577296, 0.201859236, 0.278185248, 0.16634202, 0.0324927792, 0.185975701, -0.162036508, 0.214893028, 0.144453928, 0.18897824, -0.02271723, 0.173502356, 0.0860304534, 0.157381833, -0.109898388, 0.0889903679, -0.00139595452, -0.0246559381, 0.0552617051, -0.0490884259, 0.0221240669, -0.00970905647, 0.271192163, 0.0836053491, 0.136748031, 0.0590723492, 0.131660268, -0.0782020912, 0.233400002, 0.020858407, -0.199875951, -0.10958828, -0.0476728119, -0.112283461, 0.0634761229, -0.11828354, -0.206033915, 0.193904743, 0.208372578, -0.0133872097, 0.128678188, -0.0611923672, -0.0264214631, -0.0343179964, 0.120693304, 0.242108658, -0.123052984, 0.00721185189, 0.0428376906, 0.185159311, 0.189356312, -0.121340357, -0.0659567639, 0.0139191207, -0.172991693, 0.231255203, -0.0546388291, -0.12772809, -0.186477616, -0.0920270532, -0.131607428, -0.115861528, 0.102707088, 0.152410567, 0.159929469, 0.0160477627, -0.0876519978, 0.0969803855, -0.213091269, 0.196864411, 0.273380667, -0.188008323, -0.0920328945, 0.289578468, -0.0528584607, -0.0977249518, -0.00144148862, -0.179536566, -0.0322223529, -0.212180287, 0.231571823, -0.193322748, 0.215044737, -0.0583524294, -0.148938805, -0.104199901, 0.0954470932, -0.0519888364, -0.120300457, 0.0400745571, -0.208074585, 0.16796045, -0.126946077, 0.105555303, -0.179807782, -0.139423996, -0.110121422, -0.143779054, 0.0281973183, -0.213963971, -0.00856938958, -0.181462109, 0.209135398, 0.0444553941, 0.212432578, -0.152585238, 0.0589921027, -0.0956718326, -0.202689767, 0.189238891, -0.00226314366, 0.00328245759, -0.07723362, 0.0444654375, -0.110938296, 0.11733903, 0.118250266, 0.0411194339, -0.0846743733, -0.214066923, 0.13189514, -0.14326416, -0.171151295, 0.00388705614, 0.208343133, 0.0269903056, 0.059002623, 0.0961068422, 0.100626692, 0.0702101141, 0.020035034, -0.0141857117, 0.0257037412, -0.0787355751, 0.149851128, -0.0874555111, 0.0847222954, -0.203368247, 0.0913478732, -0.190981388, 0.0381076187, -0.0793296993, -0.0151991285, 0.0998160616, -0.113543928, 0.0162660182, 0.103863224, 0.0264875349, 0.0567879528, -0.0818504989, -0.174385443, -0.00410155952, 0.0188013464, -0.0961839706, -0.133884028, -0.0904380009, -0.123644434, -0.132027194, -0.0969853327, 0.178106606, -0.164912462, -0.129356861, 0.254577816, -0.244255126, 0.085457325, -0.20408611, -0.0806175619, 0.049568817, -0.0337973684, 0.0333623476, 0.147425145, 0.115208894, -0.0453046039, 0.300857335, 0.0715077147, 0.0815929845, 0.217304617, 0.174860537, -0.217734858, -0.0545187891, -0.110197, 0.0350490846, -0.187146857, -0.0842425302, -0.155964121, 0.00266452134, -0.0114788301, -0.0303328782, -0.183492959, 0.043718189, 0.119714215, -0.0836073384, 0.194770262, 0.176857576, -0.0258767977, 0.260465145, 0.108764701, -0.0949423462, 0.0376914777, 0.063421309, 0.0491331071, 0.185503632, -0.00521813333, -0.195495903, -0.131301835, 0.135766819, -0.212390468, 0.0454258732, 0.116974734, -0.0042796433, -0.0877883956, -0.0176164117, 0.116867885, 0.084963426, -0.145454615, -0.00281196297, 0.158816293, 0.261381388, -0.103646547, -0.0409106165, 0.119343556, 0.0541383289, -0.179490834, -0.226963773, 0.0730867088, -0.0670445934, -0.146837354, -0.100336365, -0.206874445, -0.147349969, -0.0639766306, -0.0242820475, -0.0191500783, 0.0574500002, -0.118401602, -0.0355735309, -0.0470449142, 0.0599663332, -0.176558927, 0.00412532967, 0.213447168, -0.010397274, -0.0719934478, -0.0328418612, -0.00671752123, -0.0474058241, 0.162177995, -0.0395350344, 0.200220659, -0.0697177351, -0.161850125, 0.107072055, 0.178566739, 0.209856763, -0.148664251, 0.0821418315, -0.125930011, -0.173101038, 0.0771152675, 0.0780660436, -0.134412229, 0.186319694, 0.0190821849, -0.23414728, -0.104899429, 0.19066, -0.0627585649, -0.169341192, -0.178378239, -0.0991300195, -0.0998610705, 0.131659567, -0.00676505361, 0.211450562, 0.0258109439, 0.220644847, -0.207787529, 0.0453971066, 0.0513934791, 0.0972999409, 0.0140249133, 0.185306981, 0.132868722, -0.124948919, -0.0208617114, -0.0660538822, -0.103338204, 0.0198297929];
